LIN {X 0,Y 632.529,Z 1162.181,A -85,B 0,C 180,E1 6544.101,E2 6544.101} C_VEL
LIN {X 0,Y 629.019,Z 1204.643,A -85,B 0,C 180,E1 6550.428,E2 6550.428} C_VEL
LIN {X 0,Y 627.402,Z 1233.315,A -85,B 0,C 180,E1 6556.71,E2 6556.71} C_VEL
LIN {X 0,Y 626.919,Z 1250.593,A -85,B 0,C 180,E1 6563.045,E2 6563.045} C_VEL
LIN {X 0,Y 626.986,Z 1256.412,A -85,B 0,C 180,E1 6567.918,E2 6567.918} C_VEL
LIN {X 0,Y 627.218,Z 1255.317,A -85,B 0,C 180,E1 6573.469,E2 6573.469} C_VEL
LIN {X 0,Y 627.216,Z 1244.04,A -85,B 0,C 180,E1 6579.754,E2 6579.754} C_VEL
LIN {X 0,Y 628.041,Z 1219.84,A -85,B 0,C 180,E1 6586.5,E2 6586.5} C_VEL
LIN {X 0,Y 630.682,Z 1183.615,A -85,B 0,C 180,E1 6592.9,E2 6592.9} C_VEL
LIN {X 0,Y 635.527,Z 1132.969,A -85,B 0,C 180,E1 6599.124,E2 6599.124} C_VEL
LIN {X 0,Y 642.274,Z 1070.411,A -85,B 0,C 180,E1 6604.511,E2 6604.511} C_VEL
LIN {X 0,Y 649.326,Z 1000.53,A -85,B 0,C 180,E1 6608.612,E2 6608.612} C_VEL
LIN {X 0,Y 654.879,Z 926.452,A -85,B 0,C 180,E1 6611.351,E2 6611.351} C_VEL
LIN {X 0,Y 655.116,Z 892.167,A -85,B 0,C 180,E1 6612.26,E2 6612.26} C_VEL
LIN {X 0,Y 626.271,Z 839.06,A -85,B 0,C 180,E1 6615.936,E2 6615.936} C_VEL
LIN {X 0,Y 626.249,Z 839.06,A -85,B 0,C 180,E1 6624.3,E2 6624.3} C_VEL
LIN {X 0,Y 626.373,Z 839.06,A -85,B 0,C 180,E1 6632.206,E2 6632.206} C_VEL
LIN {X 0,Y 626.221,Z 839.06,A -85,B 0,C 180,E1 6640.951,E2 6640.951} C_VEL
LIN {X 0,Y 626.965,Z 839.06,A -85,B 0,C 180,E1 6649.584,E2 6649.584} C_VEL
LIN {X 0,Y 627.516,Z 839.06,A -85,B 0,C 180,E1 6659.347,E2 6659.347} C_VEL
LIN {X 0,Y 626.832,Z 839.06,A -85,B 0,C 180,E1 6667.69,E2 6667.69} C_VEL
LIN {X 0,Y 626.275,Z 839.06,A -85,B 0,C 180,E1 6676.766,E2 6676.766} C_VEL
LIN {X 0,Y 626.335,Z 839.06,A -85,B 0,C 180,E1 6685.126,E2 6685.126} C_VEL
LIN {X 0,Y 626.126,Z 839.06,A -85,B 0,C 180,E1 6693.229,E2 6693.229} C_VEL
LIN {X 0,Y 626.05,Z 839.06,A -85,B 0,C 180,E1 6701.847,E2 6701.847} C_VEL
LIN {X 0,Y 626.572,Z 841.021,A -85,B 0,C 180,E1 6703.843,E2 6703.843} C_VEL
LIN {X 0,Y 640.02,Z 863.387,A -85,B 0,C 180,E1 6705.418,E2 6705.418} C_VEL
LIN {X 0,Y 644.521,Z 885.503,A -85,B 0,C 180,E1 6706.146,E2 6706.146} C_VEL
LIN {X 0,Y 651.275,Z 900.392,A -85,B 0,C 180,E1 6706.954,E2 6706.954} C_VEL
LIN {X 0,Y 647.369,Z 977.205,A -85,B 0,C 180,E1 6708.756,E2 6708.756} C_VEL
LIN {X 0,Y 641.012,Z 1049.358,A -85,B 0,C 180,E1 6711.835,E2 6711.835} C_VEL
LIN {X 0,Y 633.382,Z 1117.843,A -85,B 0,C 180,E1 6716.34,E2 6716.34} C_VEL
LIN {X 0,Y 626.55,Z 1177.833,A -85,B 0,C 180,E1 6722.084,E2 6722.084} C_VEL
LIN {X 0,Y 621.952,Z 1224.147,A -85,B 0,C 180,E1 6728.397,E2 6728.397} C_VEL
LIN {X 0,Y 619.792,Z 1256.235,A -85,B 0,C 180,E1 6734.734,E2 6734.734} C_VEL
LIN {X 0,Y 619.023,Z 1276.005,A -85,B 0,C 180,E1 6740.828,E2 6740.828} C_VEL
LIN {X 0,Y 618.825,Z 1285.35,A -85,B 0,C 180,E1 6746.484,E2 6746.484} C_VEL
LIN {X 0,Y 618.751,Z 1286.379,A -85,B 0,C 180,E1 6752.11,E2 6752.11} C_VEL
LIN {X 0,Y 618.913,Z 1279.146,A -85,B 0,C 180,E1 6757.754,E2 6757.754} C_VEL
LIN {X 0,Y 619.502,Z 1261.052,A -85,B 0,C 180,E1 6764.027,E2 6764.027} C_VEL
LIN {X 0,Y 621.388,Z 1231.04,A -85,B 0,C 180,E1 6770.441,E2 6770.441} C_VEL
LIN {X 0,Y 625.557,Z 1187.146,A -85,B 0,C 180,E1 6776.825,E2 6776.825} C_VEL
LIN {X 0,Y 632.04,Z 1129.362,A -85,B 0,C 180,E1 6782.714,E2 6782.714} C_VEL
LIN {X 0,Y 639.563,Z 1062.77,A -85,B 0,C 180,E1 6787.421,E2 6787.421} C_VEL
LIN {X 0,Y 646.292,Z 992.668,A -85,B 0,C 180,E1 6790.706,E2 6790.706} C_VEL
LIN {X 0,Y 650.782,Z 919.257,A -85,B 0,C 180,E1 6792.72,E2 6792.72} C_VEL
LIN {X 0,Y 650.036,Z 895.654,A -85,B 0,C 180,E1 6793.232,E2 6793.232} C_VEL
LIN {X 0,Y 618.189,Z 839.06,A -85,B 0,C 180,E1 6797.021,E2 6797.021} C_VEL
LIN {X 0,Y 618.365,Z 839.06,A -85,B 0,C 180,E1 6805.331,E2 6805.331} C_VEL
LIN {X 0,Y 618.596,Z 839.06,A -85,B 0,C 180,E1 6813.607,E2 6813.607} C_VEL
LIN {X 0,Y 618.576,Z 839.06,A -85,B 0,C 180,E1 6823.575,E2 6823.575} C_VEL
LIN {X 0,Y 618.896,Z 839.06,A -85,B 0,C 180,E1 6832.211,E2 6832.211} C_VEL
LIN {X 0,Y 618.875,Z 839.06,A -85,B 0,C 180,E1 6840.662,E2 6840.662} C_VEL
LIN {X 0,Y 618.452,Z 839.06,A -85,B 0,C 180,E1 6849.135,E2 6849.135} C_VEL
LIN {X 0,Y 618.386,Z 839.06,A -85,B 0,C 180,E1 6856.346,E2 6856.346} C_VEL
LIN {X 0,Y 618.266,Z 839.06,A -85,B 0,C 180,E1 6865.387,E2 6865.387} C_VEL
LIN {X 0,Y 618.098,Z 839.06,A -85,B 0,C 180,E1 6873.476,E2 6873.476} C_VEL
LIN {X 0,Y 618.165,Z 839.06,A -85,B 0,C 180,E1 6882.395,E2 6882.395} C_VEL
LIN {X 0,Y 618.334,Z 840.427,A -85,B 0,C 180,E1 6883.456,E2 6883.456} C_VEL
LIN {X 0,Y 650.507,Z 899.763,A -85,B 0,C 180,E1 6887.454,E2 6887.454} C_VEL
LIN {X 0,Y 645.669,Z 969.285,A -85,B 0,C 180,E1 6889.502,E2 6889.502} C_VEL
LIN {X 0,Y 638.674,Z 1040.727,A -85,B 0,C 180,E1 6893.01,E2 6893.01} C_VEL
LIN {X 0,Y 631.057,Z 1107.355,A -85,B 0,C 180,E1 6897.944,E2 6897.944} C_VEL
LIN {X 0,Y 624.785,Z 1164.218,A -85,B 0,C 180,E1 6904.026,E2 6904.026} C_VEL
LIN {X 0,Y 621.153,Z 1205.493,A -85,B 0,C 180,E1 6910.33,E2 6910.33} C_VEL
LIN {X 0,Y 619.342,Z 1234.621,A -85,B 0,C 180,E1 6916.895,E2 6916.895} C_VEL
LIN {X 0,Y 618.993,Z 1250.188,A -85,B 0,C 180,E1 6922.736,E2 6922.736} C_VEL
LIN {X 0,Y 618.99,Z 1256.411,A -85,B 0,C 180,E1 6927.891,E2 6927.891} C_VEL
LIN {X 0,Y 619.195,Z 1255.317,A -85,B 0,C 180,E1 6933.514,E2 6933.514} C_VEL
LIN {X 0,Y 619.187,Z 1244.041,A -85,B 0,C 180,E1 6939.882,E2 6939.882} C_VEL
LIN {X 0,Y 620.112,Z 1221.406,A -85,B 0,C 180,E1 6946.351,E2 6946.351} C_VEL
LIN {X 0,Y 622.85,Z 1185.248,A -85,B 0,C 180,E1 6952.953,E2 6952.953} C_VEL
LIN {X 0,Y 628.001,Z 1134.743,A -85,B 0,C 180,E1 6959.309,E2 6959.309} C_VEL
LIN {X 0,Y 635.169,Z 1072.5,A -85,B 0,C 180,E1 6964.782,E2 6964.782} C_VEL
LIN {X 0,Y 642.527,Z 1004.298,A -85,B 0,C 180,E1 6968.883,E2 6968.883} C_VEL
LIN {X 0,Y 648.507,Z 930.181,A -85,B 0,C 180,E1 6971.721,E2 6971.721} C_VEL
LIN {X 0,Y 649.203,Z 895.835,A -85,B 0,C 180,E1 6972.652,E2 6972.652} C_VEL
LIN {X 0,Y 618.208,Z 839.06,A -85,B 0,C 180,E1 6976.602,E2 6976.602} C_VEL
LIN {X 0,Y 618.164,Z 839.06,A -85,B 0,C 180,E1 6985.356,E2 6985.356} C_VEL
LIN {X 0,Y 618.224,Z 839.06,A -85,B 0,C 180,E1 6993.675,E2 6993.675} C_VEL
LIN {X 0,Y 618.253,Z 839.06,A -85,B 0,C 180,E1 7002.179,E2 7002.179} C_VEL
LIN {X 0,Y 619.084,Z 839.06,A -85,B 0,C 180,E1 7010.875,E2 7010.875} C_VEL
LIN {X 0,Y 619.506,Z 839.06,A -85,B 0,C 180,E1 7019.339,E2 7019.339} C_VEL
LIN {X 0,Y 618.8,Z 839.06,A -85,B 0,C 180,E1 7027.791,E2 7027.791} C_VEL
LIN {X 0,Y 618.364,Z 839.06,A -85,B 0,C 180,E1 7036.431,E2 7036.431} C_VEL
LIN {X 0,Y 618.275,Z 839.06,A -85,B 0,C 180,E1 7045.476,E2 7045.476} C_VEL
LIN {X 0,Y 618.098,Z 839.06,A -85,B 0,C 180,E1 7053.573,E2 7053.573} C_VEL
LIN {X 0,Y 618.125,Z 839.06,A -85,B 0,C 180,E1 7062.508,E2 7062.508} C_VEL
LIN {X 0,Y 618.588,Z 841.588,A -85,B 0,C 180,E1 7063.083,E2 7063.083} C_VEL
LIN {X 0,Y 644.521,Z 885.503,A -85,B 0,C 180,E1 7066.146,E2 7066.146} C_VEL
LIN {X 0,Y 646.583,Z 902.081,A -85,B 0,C 180,E1 7066.594,E2 7066.594} C_VEL
LIN {X 0,Y 644.57,Z 920.711,A -85,B 0,C 180,E1 7066.802,E2 7066.802} C_VEL
LIN {X 0,Y 639.122,Z 999.805,A -85,B 0,C 180,E1 7069.069,E2 7069.069} C_VEL
LIN {X 0,Y 631.66,Z 1073.992,A -85,B 0,C 180,E1 7072.805,E2 7072.805} C_VEL
LIN {X 0,Y 623.945,Z 1139.278,A -85,B 0,C 180,E1 7077.768,E2 7077.768} C_VEL
LIN {X 0,Y 617.63,Z 1194.659,A -85,B 0,C 180,E1 7083.808,E2 7083.808} C_VEL
LIN {X 0,Y 613.673,Z 1237.403,A -85,B 0,C 180,E1 7090.491,E2 7090.491} C_VEL
LIN {X 0,Y 611.854,Z 1267.958,A -85,B 0,C 180,E1 7097.825,E2 7097.825} C_VEL
LIN {X 0,Y 611.014,Z 1283.797,A -85,B 0,C 180,E1 7105.012,E2 7105.012} C_VEL
LIN {X 0,Y 611.015,Z 1286.837,A -85,B 0,C 180,E1 7110.712,E2 7110.712} C_VEL
LIN {X 0,Y 610.942,Z 1280.509,A -85,B 0,C 180,E1 7117.138,E2 7117.138} C_VEL
LIN {X 0,Y 611.463,Z 1263.143,A -85,B 0,C 180,E1 7123.643,E2 7123.643} C_VEL
LIN {X 0,Y 613.267,Z 1234.809,A -85,B 0,C 180,E1 7130.019,E2 7130.019} C_VEL
LIN {X 0,Y 617.386,Z 1193.464,A -85,B 0,C 180,E1 7136.364,E2 7136.364} C_VEL
LIN {X 0,Y 624.114,Z 1136.467,A -85,B 0,C 180,E1 7142.497,E2 7142.497} C_VEL
LIN {X 0,Y 632.198,Z 1069.94,A -85,B 0,C 180,E1 7147.443,E2 7147.443} C_VEL
LIN {X 0,Y 639.445,Z 1000.576,A -85,B 0,C 180,E1 7150.87,E2 7150.87} C_VEL
LIN {X 0,Y 644.506,Z 926.944,A -85,B 0,C 180,E1 7153.057,E2 7153.057} C_VEL
LIN {X 0,Y 644.183,Z 899.082,A -85,B 0,C 180,E1 7153.661,E2 7153.661} C_VEL
LIN {X 0,Y 610.104,Z 839.06,A -85,B 0,C 180,E1 7157.851,E2 7157.851} C_VEL
LIN {X 0,Y 610.384,Z 839.06,A -85,B 0,C 180,E1 7166.429,E2 7166.429} C_VEL
LIN {X 0,Y 610.523,Z 839.06,A -85,B 0,C 180,E1 7175.177,E2 7175.177} C_VEL
LIN {X 0,Y 610.474,Z 839.06,A -85,B 0,C 180,E1 7184.831,E2 7184.831} C_VEL
LIN {X 0,Y 610.556,Z 839.06,A -85,B 0,C 180,E1 7193.539,E2 7193.539} C_VEL
LIN {X 0,Y 610.866,Z 839.06,A -85,B 0,C 180,E1 7200.671,E2 7200.671} C_VEL
LIN {X 0,Y 610.864,Z 839.06,A -85,B 0,C 180,E1 7207.81,E2 7207.81} C_VEL
LIN {X 0,Y 610.285,Z 839.06,A -85,B 0,C 180,E1 7216.721,E2 7216.721} C_VEL
LIN {X 0,Y 610.235,Z 839.06,A -85,B 0,C 180,E1 7225.746,E2 7225.746} C_VEL
LIN {X 0,Y 610.108,Z 839.06,A -85,B 0,C 180,E1 7233.973,E2 7233.973} C_VEL
LIN {X 0,Y 610.414,Z 840.999,A -85,B 0,C 180,E1 7242.67,E2 7242.67} C_VEL
LIN {X 0,Y 644.471,Z 901.549,A -85,B 0,C 180,E1 7247.003,E2 7247.003} C_VEL
LIN {X 0,Y 639.37,Z 970.596,A -85,B 0,C 180,E1 7249.08,E2 7249.08} C_VEL
LIN {X 0,Y 631.998,Z 1041.381,A -85,B 0,C 180,E1 7252.599,E2 7252.599} C_VEL
LIN {X 0,Y 623.815,Z 1108.393,A -85,B 0,C 180,E1 7257.629,E2 7257.629} C_VEL
LIN {X 0,Y 617.269,Z 1164.261,A -85,B 0,C 180,E1 7263.693,E2 7263.693} C_VEL
LIN {X 0,Y 613.256,Z 1206.563,A -85,B 0,C 180,E1 7270.271,E2 7270.271} C_VEL
LIN {X 0,Y 611.419,Z 1234.62,A -85,B 0,C 180,E1 7276.722,E2 7276.722} C_VEL
LIN {X 0,Y 611.016,Z 1250.187,A -85,B 0,C 180,E1 7282.641,E2 7282.641} C_VEL
LIN {X 0,Y 610.994,Z 1256.411,A -85,B 0,C 180,E1 7287.864,E2 7287.864} C_VEL
LIN {X 0,Y 611.174,Z 1255.317,A -85,B 0,C 180,E1 7293.56,E2 7293.56} C_VEL
LIN {X 0,Y 611.169,Z 1244.042,A -85,B 0,C 180,E1 7300.013,E2 7300.013} C_VEL
LIN {X 0,Y 612.17,Z 1221.41,A -85,B 0,C 180,E1 7306.57,E2 7306.57} C_VEL
LIN {X 0,Y 615.056,Z 1186.459,A -85,B 0,C 180,E1 7313.068,E2 7313.068} C_VEL
LIN {X 0,Y 620.57,Z 1135.75,A -85,B 0,C 180,E1 7319.58,E2 7319.58} C_VEL
LIN {X 0,Y 628.092,Z 1074.411,A -85,B 0,C 180,E1 7325.072,E2 7325.072} C_VEL
LIN {X 0,Y 635.917,Z 1006.392,A -85,B 0,C 180,E1 7329.244,E2 7329.244} C_VEL
LIN {X 0,Y 642.356,Z 932.017,A -85,B 0,C 180,E1 7332.149,E2 7332.149} C_VEL
LIN {X 0,Y 643.12,Z 899.03,A -85,B 0,C 180,E1 7333.078,E2 7333.078} C_VEL
LIN {X 0,Y 610.158,Z 839.06,A -85,B 0,C 180,E1 7337.417,E2 7337.417} C_VEL
LIN {X 0,Y 610.114,Z 839.06,A -85,B 0,C 180,E1 7346.466,E2 7346.466} C_VEL
LIN {X 0,Y 610.263,Z 839.06,A -85,B 0,C 180,E1 7355.228,E2 7355.228} C_VEL
LIN {X 0,Y 610.445,Z 839.06,A -85,B 0,C 180,E1 7363.435,E2 7363.435} C_VEL
LIN {X 0,Y 610.9,Z 839.06,A -85,B 0,C 180,E1 7372.19,E2 7372.19} C_VEL
LIN {X 0,Y 610.764,Z 839.06,A -85,B 0,C 180,E1 7380.753,E2 7380.753} C_VEL
LIN {X 0,Y 610.749,Z 839.06,A -85,B 0,C 180,E1 7387.894,E2 7387.894} C_VEL
LIN {X 0,Y 610.296,Z 839.06,A -85,B 0,C 180,E1 7396.728,E2 7396.728} C_VEL
LIN {X 0,Y 610.285,Z 839.06,A -85,B 0,C 180,E1 7404.776,E2 7404.776} C_VEL
LIN {X 0,Y 610.117,Z 839.06,A -85,B 0,C 180,E1 7413.535,E2 7413.535} C_VEL
LIN {X 0,Y 610.295,Z 840.83,A -85,B 0,C 180,E1 7422.238,E2 7422.238} C_VEL
LIN {X 0,Y 645.268,Z 901.082,A -85,B 0,C 180,E1 7426.466,E2 7426.466} C_VEL
LIN {X 0,Y 644.57,Z 920.711,A -85,B 0,C 180,E1 7426.802,E2 7426.802} C_VEL
LIN {X 0,Y 637.098,Z 955.226,A -85,B 0,C 180,E1 7427.137,E2 7427.137} C_VEL
LIN {X 0,Y 630.637,Z 1026.622,A -85,B 0,C 180,E1 7429.756,E2 7429.756} C_VEL
LIN {X 0,Y 622.159,Z 1097.78,A -85,B 0,C 180,E1 7433.945,E2 7433.945} C_VEL
LIN {X 0,Y 614.134,Z 1160.209,A -85,B 0,C 180,E1 7439.391,E2 7439.391} C_VEL
LIN {X 0,Y 608.038,Z 1211.489,A -85,B 0,C 180,E1 7445.807,E2 7445.807} C_VEL
LIN {X 0,Y 604.534,Z 1249.804,A -85,B 0,C 180,E1 7452.784,E2 7452.784} C_VEL
LIN {X 0,Y 603.318,Z 1272.228,A -85,B 0,C 180,E1 7459.122,E2 7459.122} C_VEL
LIN {X 0,Y 603.036,Z 1283.794,A -85,B 0,C 180,E1 7464.945,E2 7464.945} C_VEL
LIN {X 0,Y 603.01,Z 1286.837,A -85,B 0,C 180,E1 7470.722,E2 7470.722} C_VEL
LIN {X 0,Y 602.961,Z 1280.508,A -85,B 0,C 180,E1 7477.233,E2 7477.233} C_VEL
LIN {X 0,Y 603.513,Z 1263.143,A -85,B 0,C 180,E1 7483.826,E2 7483.826} C_VEL
LIN {X 0,Y 605.407,Z 1235.634,A -85,B 0,C 180,E1 7490.131,E2 7490.131} C_VEL
LIN {X 0,Y 609.837,Z 1193.617,A -85,B 0,C 180,E1 7496.695,E2 7496.695} C_VEL
LIN {X 0,Y 616.905,Z 1137.661,A -85,B 0,C 180,E1 7502.806,E2 7502.806} C_VEL
LIN {X 0,Y 625.495,Z 1071.067,A -85,B 0,C 180,E1 7507.834,E2 7507.834} C_VEL
LIN {X 0,Y 633.192,Z 1001.774,A -85,B 0,C 180,E1 7511.306,E2 7511.306} C_VEL
LIN {X 0,Y 638.628,Z 927.423,A -85,B 0,C 180,E1 7513.539,E2 7513.539} C_VEL
LIN {X 0,Y 638.377,Z 902.376,A -85,B 0,C 180,E1 7514.1,E2 7514.1} C_VEL
LIN {X 0,Y 602.069,Z 839.06,A -85,B 0,C 180,E1 7518.711,E2 7518.711} C_VEL
LIN {X 0,Y 602.468,Z 839.06,A -85,B 0,C 180,E1 7527.581,E2 7527.581} C_VEL
LIN {X 0,Y 602.512,Z 839.06,A -85,B 0,C 180,E1 7535.404,E2 7535.404} C_VEL
LIN {X 0,Y 602.456,Z 839.06,A -85,B 0,C 180,E1 7544.624,E2 7544.624} C_VEL
LIN {X 0,Y 602.594,Z 839.06,A -85,B 0,C 180,E1 7553.453,E2 7553.453} C_VEL
LIN {X 0,Y 602.858,Z 839.06,A -85,B 0,C 180,E1 7560.68,E2 7560.68} C_VEL
LIN {X 0,Y 602.831,Z 839.06,A -85,B 0,C 180,E1 7567.915,E2 7567.915} C_VEL
LIN {X 0,Y 602.28,Z 839.06,A -85,B 0,C 180,E1 7576.796,E2 7576.796} C_VEL
LIN {X 0,Y 602.317,Z 839.06,A -85,B 0,C 180,E1 7584.513,E2 7584.513} C_VEL
LIN {X 0,Y 602.127,Z 839.06,A -85,B 0,C 180,E1 7592.753,E2 7592.753} C_VEL
LIN {X 0,Y 602.079,Z 839.139,A -85,B 0,C 180,E1 7601.764,E2 7601.764} C_VEL
LIN {X 0,Y 638.349,Z 904.917,A -85,B 0,C 180,E1 7606.582,E2 7606.582} C_VEL
LIN {X 0,Y 632.904,Z 973.934,A -85,B 0,C 180,E1 7608.728,E2 7608.728} C_VEL
LIN {X 0,Y 625.101,Z 1044.237,A -85,B 0,C 180,E1 7612.319,E2 7612.319} C_VEL
LIN {X 0,Y 616.454,Z 1110.841,A -85,B 0,C 180,E1 7617.438,E2 7617.438} C_VEL
LIN {X 0,Y 609.485,Z 1166.513,A -85,B 0,C 180,E1 7623.638,E2 7623.638} C_VEL
LIN {X 0,Y 605.361,Z 1207.623,A -85,B 0,C 180,E1 7630.211,E2 7630.211} C_VEL
LIN {X 0,Y 603.395,Z 1235.781,A -85,B 0,C 180,E1 7636.912,E2 7636.912} C_VEL
LIN {X 0,Y 602.915,Z 1251.796,A -85,B 0,C 180,E1 7643.494,E2 7643.494} C_VEL
LIN {X 0,Y 602.68,Z 1256.848,A -85,B 0,C 180,E1 7649.278,E2 7649.278} C_VEL
LIN {X 0,Y 602.912,Z 1252.806,A -85,B 0,C 180,E1 7655.78,E2 7655.78} C_VEL
LIN {X 0,Y 603.585,Z 1236.661,A -85,B 0,C 180,E1 7662.713,E2 7662.713} C_VEL
LIN {X 0,Y 605.898,Z 1205.828,A -85,B 0,C 180,E1 7670.032,E2 7670.032} C_VEL
LIN {X 0,Y 610.609,Z 1160.875,A -85,B 0,C 180,E1 7676.987,E2 7676.987} C_VEL
LIN {X 0,Y 617.438,Z 1104.611,A -85,B 0,C 180,E1 7683.033,E2 7683.033} C_VEL
LIN {X 0,Y 625.742,Z 1038.363,A -85,B 0,C 180,E1 7687.965,E2 7687.965} C_VEL
LIN {X 0,Y 633.664,Z 964.987,A -85,B 0,C 180,E1 7691.542,E2 7691.542} C_VEL
LIN {X 0,Y 637.241,Z 902.506,A -85,B 0,C 180,E1 7693.491,E2 7693.491} C_VEL
LIN {X 0,Y 603.882,Z 844.033,A -85,B 0,C 180,E1 7697.868,E2 7697.868} C_VEL
LIN {X 0,Y 602.111,Z 839.06,A -85,B 0,C 180,E1 7698.163,E2 7698.163} C_VEL
LIN {X 0,Y 602.125,Z 839.06,A -85,B 0,C 180,E1 7707.247,E2 7707.247} C_VEL
LIN {X 0,Y 602.303,Z 839.06,A -85,B 0,C 180,E1 7715.486,E2 7715.486} C_VEL
LIN {X 0,Y 602.666,Z 839.06,A -85,B 0,C 180,E1 7724.716,E2 7724.716} C_VEL
LIN {X 0,Y 602.908,Z 839.06,A -85,B 0,C 180,E1 7732.086,E2 7732.086} C_VEL
LIN {X 0,Y 602.758,Z 839.06,A -85,B 0,C 180,E1 7740.763,E2 7740.763} C_VEL
LIN {X 0,Y 602.699,Z 839.06,A -85,B 0,C 180,E1 7748,E2 7748} C_VEL
LIN {X 0,Y 602.278,Z 839.06,A -85,B 0,C 180,E1 7756.883,E2 7756.883} C_VEL
LIN {X 0,Y 602.3,Z 839.06,A -85,B 0,C 180,E1 7764.605,E2 7764.605} C_VEL
LIN {X 0,Y 602.121,Z 839.06,A -85,B 0,C 180,E1 7772.852,E2 7772.852} C_VEL
LIN {X 0,Y 602.239,Z 840.755,A -85,B 0,C 180,E1 7781.393,E2 7781.393} C_VEL
LIN {X 0,Y 639.23,Z 904.05,A -85,B 0,C 180,E1 7786.005,E2 7786.005} C_VEL
LIN {X 0,Y 637.098,Z 955.226,A -85,B 0,C 180,E1 7787.137,E2 7787.137} C_VEL
LIN {X 0,Y 628.191,Z 989.03,A -85,B 0,C 180,E1 7787.698,E2 7787.698} C_VEL
LIN {X 0,Y 620.228,Z 1061.943,A -85,B 0,C 180,E1 7791.144,E2 7791.144} C_VEL
LIN {X 0,Y 611.113,Z 1129.374,A -85,B 0,C 180,E1 7796.018,E2 7796.018} C_VEL
LIN {X 0,Y 603.289,Z 1187.108,A -85,B 0,C 180,E1 7802.094,E2 7802.094} C_VEL
LIN {X 0,Y 598.231,Z 1232.469,A -85,B 0,C 180,E1 7808.996,E2 7808.996} C_VEL
LIN {X 0,Y 596.057,Z 1264.475,A -85,B 0,C 180,E1 7816.374,E2 7816.374} C_VEL
LIN {X 0,Y 595.5,Z 1281.719,A -85,B 0,C 180,E1 7823.413,E2 7823.413} C_VEL
LIN {X 0,Y 595.032,Z 1286.837,A -85,B 0,C 180,E1 7830.731,E2 7830.731} C_VEL
LIN {X 0,Y 594.977,Z 1280.505,A -85,B 0,C 180,E1 7837.33,E2 7837.33} C_VEL
LIN {X 0,Y 595.579,Z 1263.142,A -85,B 0,C 180,E1 7844.014,E2 7844.014} C_VEL
LIN {X 0,Y 597.651,Z 1235.436,A -85,B 0,C 180,E1 7850.443,E2 7850.443} C_VEL
LIN {X 0,Y 602.302,Z 1193.887,A -85,B 0,C 180,E1 7857.018,E2 7857.018} C_VEL
LIN {X 0,Y 609.977,Z 1137.087,A -85,B 0,C 180,E1 7863.284,E2 7863.284} C_VEL
LIN {X 0,Y 618.981,Z 1071.107,A -85,B 0,C 180,E1 7868.301,E2 7868.301} C_VEL
LIN {X 0,Y 627.135,Z 1001.143,A -85,B 0,C 180,E1 7871.824,E2 7871.824} C_VEL
LIN {X 0,Y 632.778,Z 928.03,A -85,B 0,C 180,E1 7874.028,E2 7874.028} C_VEL
LIN {X 0,Y 632.297,Z 905.261,A -85,B 0,C 180,E1 7874.578,E2 7874.578} C_VEL
LIN {X 0,Y 596.01,Z 844.293,A -85,B 0,C 180,E1 7879.222,E2 7879.222} C_VEL
LIN {X 0,Y 594.085,Z 839.06,A -85,B 0,C 180,E1 7879.61,E2 7879.61} C_VEL
LIN {X 0,Y 594.467,Z 839.06,A -85,B 0,C 180,E1 7888.816,E2 7888.816} C_VEL
LIN {X 0,Y 594.331,Z 839.06,A -85,B 0,C 180,E1 7896.646,E2 7896.646} C_VEL
LIN {X 0,Y 594.359,Z 839.06,A -85,B 0,C 180,E1 7905.922,E2 7905.922} C_VEL
LIN {X 0,Y 594.602,Z 839.06,A -85,B 0,C 180,E1 7913.364,E2 7913.364} C_VEL
LIN {X 0,Y 594.849,Z 839.06,A -85,B 0,C 180,E1 7920.689,E2 7920.689} C_VEL
LIN {X 0,Y 594.782,Z 839.06,A -85,B 0,C 180,E1 7928.023,E2 7928.023} C_VEL
LIN {X 0,Y 594.225,Z 839.06,A -85,B 0,C 180,E1 7937.031,E2 7937.031} C_VEL
LIN {X 0,Y 594.243,Z 839.06,A -85,B 0,C 180,E1 7944.916,E2 7944.916} C_VEL
LIN {X 0,Y 594.024,Z 839.06,A -85,B 0,C 180,E1 7953.84,E2 7953.84} C_VEL
LIN {X 0,Y 594.3,Z 840.985,A -85,B 0,C 180,E1 7960.944,E2 7960.944} C_VEL
LIN {X 0,Y 628.756,Z 900.689,A -85,B 0,C 180,E1 7965.629,E2 7965.629} C_VEL
LIN {X 0,Y 632.023,Z 912.179,A -85,B 0,C 180,E1 7966.257,E2 7966.257} C_VEL
LIN {X 0,Y 626.061,Z 981.748,A -85,B 0,C 180,E1 7968.558,E2 7968.558} C_VEL
LIN {X 0,Y 617.713,Z 1050.945,A -85,B 0,C 180,E1 7972.276,E2 7972.276} C_VEL
LIN {X 0,Y 608.668,Z 1116.732,A -85,B 0,C 180,E1 7977.571,E2 7977.571} C_VEL
LIN {X 0,Y 601.336,Z 1171.593,A -85,B 0,C 180,E1 7983.982,E2 7983.982} C_VEL
LIN {X 0,Y 597.151,Z 1211.506,A -85,B 0,C 180,E1 7990.701,E2 7990.701} C_VEL
LIN {X 0,Y 595.367,Z 1236.942,A -85,B 0,C 180,E1 7997.108,E2 7997.108} C_VEL
LIN {X 0,Y 594.938,Z 1251.792,A -85,B 0,C 180,E1 8003.406,E2 8003.406} C_VEL
LIN {X 0,Y 594.681,Z 1256.848,A -85,B 0,C 180,E1 8009.268,E2 8009.268} C_VEL
LIN {X 0,Y 594.939,Z 1252.807,A -85,B 0,C 180,E1 8015.858,E2 8015.858} C_VEL
LIN {X 0,Y 595.685,Z 1236.664,A -85,B 0,C 180,E1 8022.885,E2 8022.885} C_VEL
LIN {X 0,Y 598.162,Z 1205.829,A -85,B 0,C 180,E1 8030.303,E2 8030.303} C_VEL
LIN {X 0,Y 603.221,Z 1160.195,A -85,B 0,C 180,E1 8037.44,E2 8037.44} C_VEL
LIN {X 0,Y 610.695,Z 1102.99,A -85,B 0,C 180,E1 8043.61,E2 8043.61} C_VEL
LIN {X 0,Y 619.491,Z 1036.605,A -85,B 0,C 180,E1 8048.546,E2 8048.546} C_VEL
LIN {X 0,Y 627.757,Z 963.177,A -85,B 0,C 180,E1 8052.108,E2 8052.108} C_VEL
LIN {X 0,Y 631.077,Z 905.613,A -85,B 0,C 180,E1 8053.936,E2 8053.936} C_VEL
LIN {X 0,Y 599.364,Z 849.392,A -85,B 0,C 180,E1 8058.257,E2 8058.257} C_VEL
LIN {X 0,Y 594.03,Z 839.06,A -85,B 0,C 180,E1 8059.198,E2 8059.198} C_VEL
LIN {X 0,Y 594.219,Z 839.06,A -85,B 0,C 180,E1 8068.488,E2 8068.488} C_VEL
LIN {X 0,Y 594.377,Z 839.06,A -85,B 0,C 180,E1 8076.739,E2 8076.739} C_VEL
LIN {X 0,Y 594.782,Z 839.06,A -85,B 0,C 180,E1 8086.019,E2 8086.019} C_VEL
LIN {X 0,Y 594.567,Z 839.06,A -85,B 0,C 180,E1 8093.449,E2 8093.449} C_VEL
LIN {X 0,Y 594.756,Z 839.06,A -85,B 0,C 180,E1 8100.773,E2 8100.773} C_VEL
LIN {X 0,Y 594.653,Z 839.06,A -85,B 0,C 180,E1 8108.109,E2 8108.109} C_VEL
LIN {X 0,Y 594.253,Z 839.06,A -85,B 0,C 180,E1 8117.118,E2 8117.118} C_VEL
LIN {X 0,Y 594.253,Z 839.06,A -85,B 0,C 180,E1 8124.961,E2 8124.961} C_VEL
LIN {X 0,Y 594.031,Z 839.06,A -85,B 0,C 180,E1 8133.843,E2 8133.843} C_VEL
LIN {X 0,Y 594.253,Z 840.855,A -85,B 0,C 180,E1 8140.521,E2 8140.521} C_VEL
LIN {X 0,Y 633.142,Z 906.971,A -85,B 0,C 180,E1 8145.528,E2 8145.528} C_VEL
LIN {X 0,Y 628.46,Z 986.241,A -85,B 0,C 180,E1 8147.604,E2 8147.604} C_VEL
LIN {X 0,Y 628.191,Z 989.03,A -85,B 0,C 180,E1 8147.698,E2 8147.698} C_VEL
LIN {X 0,Y 619.77,Z 1011.161,A -85,B 0,C 180,E1 8148.057,E2 8148.057} C_VEL
LIN {X 0,Y 610.69,Z 1083.868,A -85,B 0,C 180,E1 8152.038,E2 8152.038} C_VEL
LIN {X 0,Y 601.535,Z 1148.423,A -85,B 0,C 180,E1 8157.373,E2 8157.373} C_VEL
LIN {X 0,Y 594.154,Z 1202.648,A -85,B 0,C 180,E1 8163.849,E2 8163.849} C_VEL
LIN {X 0,Y 589.634,Z 1244.839,A -85,B 0,C 180,E1 8171.227,E2 8171.227} C_VEL
LIN {X 0,Y 587.441,Z 1272.229,A -85,B 0,C 180,E1 8178.825,E2 8178.825} C_VEL
LIN {X 0,Y 587.081,Z 1283.788,A -85,B 0,C 180,E1 8184.808,E2 8184.808} C_VEL
LIN {X 0,Y 587.027,Z 1286.837,A -85,B 0,C 180,E1 8190.741,E2 8190.741} C_VEL
LIN {X 0,Y 586.975,Z 1280.502,A -85,B 0,C 180,E1 8197.431,E2 8197.431} C_VEL
LIN {X 0,Y 587.657,Z 1263.141,A -85,B 0,C 180,E1 8204.207,E2 8204.207} C_VEL
LIN {X 0,Y 590.07,Z 1233.454,A -85,B 0,C 180,E1 8211.112,E2 8211.112} C_VEL
LIN {X 0,Y 595.727,Z 1188.276,A -85,B 0,C 180,E1 8218.129,E2 8218.129} C_VEL
LIN {X 0,Y 604.023,Z 1130.665,A -85,B 0,C 180,E1 8224.314,E2 8224.314} C_VEL
LIN {X 0,Y 613.535,Z 1063.651,A -85,B 0,C 180,E1 8229.246,E2 8229.246} C_VEL
LIN {X 0,Y 621.894,Z 993.828,A -85,B 0,C 180,E1 8232.612,E2 8232.612} C_VEL
LIN {X 0,Y 627.33,Z 922.424,A -85,B 0,C 180,E1 8234.643,E2 8234.643} C_VEL
LIN {X 0,Y 626.266,Z 908.039,A -85,B 0,C 180,E1 8235.067,E2 8235.067} C_VEL
LIN {X 0,Y 588.791,Z 845.036,A -85,B 0,C 180,E1 8240.024,E2 8240.024} C_VEL
LIN {X 0,Y 586.171,Z 839.06,A -85,B 0,C 180,E1 8240.589,E2 8240.589} C_VEL
LIN {X 0,Y 586.447,Z 839.06,A -85,B 0,C 180,E1 8250.136,E2 8250.136} C_VEL
LIN {X 0,Y 586.125,Z 839.06,A -85,B 0,C 180,E1 8257.909,E2 8257.909} C_VEL
LIN {X 0,Y 586.332,Z 839.06,A -85,B 0,C 180,E1 8266.155,E2 8266.155} C_VEL
LIN {X 0,Y 586.622,Z 839.06,A -85,B 0,C 180,E1 8273.274,E2 8273.274} C_VEL
LIN {X 0,Y 586.841,Z 839.06,A -85,B 0,C 180,E1 8280.698,E2 8280.698} C_VEL
LIN {X 0,Y 586.735,Z 839.06,A -85,B 0,C 180,E1 8288.133,E2 8288.133} C_VEL
LIN {X 0,Y 586.178,Z 839.06,A -85,B 0,C 180,E1 8297.272,E2 8297.272} C_VEL
LIN {X 0,Y 586.227,Z 839.06,A -85,B 0,C 180,E1 8305.232,E2 8305.232} C_VEL
LIN {X 0,Y 586.043,Z 839.06,A -85,B 0,C 180,E1 8313.77,E2 8313.77} C_VEL
LIN {X 0,Y 586.133,Z 840.441,A -85,B 0,C 180,E1 8319.999,E2 8319.999} C_VEL
LIN {X 0,Y 621.646,Z 901.479,A -85,B 0,C 180,E1 8324.997,E2 8324.997} C_VEL
LIN {X 0,Y 626.079,Z 914.944,A -85,B 0,C 180,E1 8325.812,E2 8325.812} C_VEL
LIN {X 0,Y 619.684,Z 984.03,A -85,B 0,C 180,E1 8328.162,E2 8328.162} C_VEL
LIN {X 0,Y 610.83,Z 1053.59,A -85,B 0,C 180,E1 8331.98,E2 8331.98} C_VEL
LIN {X 0,Y 601.338,Z 1118.473,A -85,B 0,C 180,E1 8337.321,E2 8337.321} C_VEL
LIN {X 0,Y 593.627,Z 1172.937,A -85,B 0,C 180,E1 8343.823,E2 8343.823} C_VEL
LIN {X 0,Y 589.327,Z 1211.681,A -85,B 0,C 180,E1 8350.473,E2 8350.473} C_VEL
LIN {X 0,Y 587.441,Z 1236.94,A -85,B 0,C 180,E1 8356.93,E2 8356.93} C_VEL
LIN {X 0,Y 586.961,Z 1251.788,A -85,B 0,C 180,E1 8363.316,E2 8363.316} C_VEL
LIN {X 0,Y 586.683,Z 1256.848,A -85,B 0,C 180,E1 8369.258,E2 8369.258} C_VEL
LIN {X 0,Y 586.881,Z 1253.736,A -85,B 0,C 180,E1 8375.194,E2 8375.194} C_VEL
LIN {X 0,Y 587.32,Z 1240.12,A -85,B 0,C 180,E1 8381.934,E2 8381.934} C_VEL
LIN {X 0,Y 589.119,Z 1214.638,A -85,B 0,C 180,E1 8388.79,E2 8388.79} C_VEL
LIN {X 0,Y 593.541,Z 1175.015,A -85,B 0,C 180,E1 8395.773,E2 8395.773} C_VEL
LIN {X 0,Y 600.98,Z 1120.999,A -85,B 0,C 180,E1 8402.329,E2 8402.329} C_VEL
LIN {X 0,Y 610.333,Z 1056.636,A -85,B 0,C 180,E1 8407.719,E2 8407.719} C_VEL
LIN {X 0,Y 619.42,Z 986.417,A -85,B 0,C 180,E1 8411.639,E2 8411.639} C_VEL
LIN {X 0,Y 626.039,Z 916.562,A -85,B 0,C 180,E1 8414.052,E2 8414.052} C_VEL
LIN {X 0,Y 622.509,Z 903.37,A -85,B 0,C 180,E1 8414.784,E2 8414.784} C_VEL
LIN {X 0,Y 589.079,Z 845.345,A -85,B 0,C 180,E1 8419.476,E2 8419.476} C_VEL
LIN {X 0,Y 586.009,Z 839.06,A -85,B 0,C 180,E1 8420.29,E2 8420.29} C_VEL
LIN {X 0,Y 586.25,Z 839.06,A -85,B 0,C 180,E1 8429.741,E2 8429.741} C_VEL
LIN {X 0,Y 586.344,Z 839.06,A -85,B 0,C 180,E1 8438.01,E2 8438.01} C_VEL
LIN {X 0,Y 586.75,Z 839.06,A -85,B 0,C 180,E1 8447.347,E2 8447.347} C_VEL
LIN {X 0,Y 586.384,Z 839.06,A -85,B 0,C 180,E1 8455.37,E2 8455.37} C_VEL
LIN {X 0,Y 586.75,Z 839.06,A -85,B 0,C 180,E1 8460.783,E2 8460.783} C_VEL
LIN {X 0,Y 586.608,Z 839.06,A -85,B 0,C 180,E1 8468.221,E2 8468.221} C_VEL
LIN {X 0,Y 586.199,Z 839.06,A -85,B 0,C 180,E1 8477.361,E2 8477.361} C_VEL
LIN {X 0,Y 586.203,Z 839.06,A -85,B 0,C 180,E1 8485.327,E2 8485.327} C_VEL
LIN {X 0,Y 586.029,Z 839.06,A -85,B 0,C 180,E1 8493.874,E2 8493.874} C_VEL
LIN {X 0,Y 586.321,Z 840.939,A -85,B 0,C 180,E1 8499.615,E2 8499.615} C_VEL
LIN {X 0,Y 624.852,Z 905.465,A -85,B 0,C 180,E1 8504.755,E2 8504.755} C_VEL
LIN {X 0,Y 627.452,Z 915.546,A -85,B 0,C 180,E1 8505.199,E2 8505.199} C_VEL
LIN {X 0,Y 621.618,Z 993.895,A -85,B 0,C 180,E1 8507.367,E2 8507.367} C_VEL
LIN {X 0,Y 619.77,Z 1011.161,A -85,B 0,C 180,E1 8508.057,E2 8508.057} C_VEL
LIN {X 0,Y 609.963,Z 1043.36,A -85,B 0,C 180,E1 8509.12,E2 8509.12} C_VEL
LIN {X 0,Y 600.01,Z 1111.635,A -85,B 0,C 180,E1 8513.619,E2 8513.619} C_VEL
LIN {X 0,Y 590.55,Z 1173,A -85,B 0,C 180,E1 8519.591,E2 8519.591} C_VEL
LIN {X 0,Y 583.889,Z 1221.503,A -85,B 0,C 180,E1 8526.429,E2 8526.429} C_VEL
LIN {X 0,Y 580.379,Z 1254.894,A -85,B 0,C 180,E1 8533.33,E2 8533.33} C_VEL
LIN {X 0,Y 579.111,Z 1276.005,A -85,B 0,C 180,E1 8540.19,E2 8540.19} C_VEL
LIN {X 0,Y 578.868,Z 1285.349,A -85,B 0,C 180,E1 8546.241,E2 8546.241} C_VEL
LIN {X 0,Y 578.82,Z 1286.379,A -85,B 0,C 180,E1 8552.255,E2 8552.255} C_VEL
LIN {X 0,Y 579.238,Z 1277.595,A -85,B 0,C 180,E1 8559.048,E2 8559.048} C_VEL
LIN {X 0,Y 580.977,Z 1254.689,A -85,B 0,C 180,E1 8566.705,E2 8566.705} C_VEL
LIN {X 0,Y 584.821,Z 1217.061,A -85,B 0,C 180,E1 8574.28,E2 8574.28} C_VEL
LIN {X 0,Y 591.822,Z 1165.647,A -85,B 0,C 180,E1 8581.232,E2 8581.232} C_VEL
LIN {X 0,Y 601.152,Z 1104.516,A -85,B 0,C 180,E1 8586.934,E2 8586.934} C_VEL
LIN {X 0,Y 610.899,Z 1034.056,A -85,B 0,C 180,E1 8591.38,E2 8591.38} C_VEL
LIN {X 0,Y 618.936,Z 957.216,A -85,B 0,C 180,E1 8594.351,E2 8594.351} C_VEL
LIN {X 0,Y 620.815,Z 912.065,A -85,B 0,C 180,E1 8595.491,E2 8595.491} C_VEL
LIN {X 0,Y 584.529,Z 850.775,A -85,B 0,C 180,E1 8600.413,E2 8600.413} C_VEL
LIN {X 0,Y 578.113,Z 839.06,A -85,B 0,C 180,E1 8601.558,E2 8601.558} C_VEL
LIN {X 0,Y 578.458,Z 839.06,A -85,B 0,C 180,E1 8610.924,E2 8610.924} C_VEL
LIN {X 0,Y 578.021,Z 839.06,A -85,B 0,C 180,E1 8619.2,E2 8619.2} C_VEL
LIN {X 0,Y 578.272,Z 839.06,A -85,B 0,C 180,E1 8627.07,E2 8627.07} C_VEL
LIN {X 0,Y 578.386,Z 839.06,A -85,B 0,C 180,E1 8634.689,E2 8634.689} C_VEL
LIN {X 0,Y 578.833,Z 839.06,A -85,B 0,C 180,E1 8640.708,E2 8640.708} C_VEL
LIN {X 0,Y 578.691,Z 839.06,A -85,B 0,C 180,E1 8648.247,E2 8648.247} C_VEL
LIN {X 0,Y 578.164,Z 839.06,A -85,B 0,C 180,E1 8657.519,E2 8657.519} C_VEL
LIN {X 0,Y 578.193,Z 839.06,A -85,B 0,C 180,E1 8665.608,E2 8665.608} C_VEL
LIN {X 0,Y 578.016,Z 839.06,A -85,B 0,C 180,E1 8674.304,E2 8674.304} C_VEL
LIN {X 0,Y 578.209,Z 840.785,A -85,B 0,C 180,E1 8679.053,E2 8679.053} C_VEL
LIN {X 0,Y 615.112,Z 903.174,A -85,B 0,C 180,E1 8684.422,E2 8684.422} C_VEL
LIN {X 0,Y 620.082,Z 918.824,A -85,B 0,C 180,E1 8685.385,E2 8685.385} C_VEL
LIN {X 0,Y 613.08,Z 988.633,A -85,B 0,C 180,E1 8687.861,E2 8687.861} C_VEL
LIN {X 0,Y 603.856,Z 1056.414,A -85,B 0,C 180,E1 8691.695,E2 8691.695} C_VEL
LIN {X 0,Y 594.008,Z 1120.207,A -85,B 0,C 180,E1 8697.064,E2 8697.064} C_VEL
LIN {X 0,Y 585.909,Z 1174.336,A -85,B 0,C 180,E1 8703.67,E2 8703.67} C_VEL
LIN {X 0,Y 581.318,Z 1213.498,A -85,B 0,C 180,E1 8710.602,E2 8710.602} C_VEL
LIN {X 0,Y 579.413,Z 1238.088,A -85,B 0,C 180,E1 8717.131,E2 8717.131} C_VEL
LIN {X 0,Y 578.948,Z 1252.778,A -85,B 0,C 180,E1 8723.868,E2 8723.868} C_VEL
LIN {X 0,Y 579.036,Z 1256.827,A -85,B 0,C 180,E1 8730.751,E2 8730.751} C_VEL
LIN {X 0,Y 579.473,Z 1249.059,A -85,B 0,C 180,E1 8738.284,E2 8738.284} C_VEL
LIN {X 0,Y 580.412,Z 1227.584,A -85,B 0,C 180,E1 8745.94,E2 8745.94} C_VEL
LIN {X 0,Y 583.884,Z 1191.855,A -85,B 0,C 180,E1 8753.466,E2 8753.466} C_VEL
LIN {X 0,Y 590.669,Z 1142.33,A -85,B 0,C 180,E1 8760.439,E2 8760.439} C_VEL
LIN {X 0,Y 600.125,Z 1081.182,A -85,B 0,C 180,E1 8766.368,E2 8766.368} C_VEL
LIN {X 0,Y 609.925,Z 1013.604,A -85,B 0,C 180,E1 8770.823,E2 8770.823} C_VEL
LIN {X 0,Y 618.161,Z 939.664,A -85,B 0,C 180,E1 8773.945,E2 8773.945} C_VEL
LIN {X 0,Y 619.092,Z 912.151,A -85,B 0,C 180,E1 8774.827,E2 8774.827} C_VEL
LIN {X 0,Y 589.037,Z 857.554,A -85,B 0,C 180,E1 8779.256,E2 8779.256} C_VEL
LIN {X 0,Y 578.017,Z 839.06,A -85,B 0,C 180,E1 8781.022,E2 8781.022} C_VEL
LIN {X 0,Y 578.161,Z 839.06,A -85,B 0,C 180,E1 8789.272,E2 8789.272} C_VEL
LIN {X 0,Y 578.279,Z 839.06,A -85,B 0,C 180,E1 8798.741,E2 8798.741} C_VEL
LIN {X 0,Y 578.738,Z 839.06,A -85,B 0,C 180,E1 8807.169,E2 8807.169} C_VEL
LIN {X 0,Y 578.391,Z 839.06,A -85,B 0,C 180,E1 8814.776,E2 8814.776} C_VEL
LIN {X 0,Y 578.743,Z 839.06,A -85,B 0,C 180,E1 8820.794,E2 8820.794} C_VEL
LIN {X 0,Y 578.567,Z 839.06,A -85,B 0,C 180,E1 8828.336,E2 8828.336} C_VEL
LIN {X 0,Y 578.153,Z 839.06,A -85,B 0,C 180,E1 8837.61,E2 8837.61} C_VEL
LIN {X 0,Y 578.187,Z 839.06,A -85,B 0,C 180,E1 8845.704,E2 8845.704} C_VEL
LIN {X 0,Y 578.006,Z 839.06,A -85,B 0,C 180,E1 8854.409,E2 8854.409} C_VEL
LIN {X 0,Y 578.251,Z 840.776,A -85,B 0,C 180,E1 8858.645,E2 8858.645} C_VEL
LIN {X 0,Y 618.048,Z 906.725,A -85,B 0,C 180,E1 8864.146,E2 8864.146} C_VEL
LIN {X 0,Y 621.59,Z 918.098,A -85,B 0,C 180,E1 8864.731,E2 8864.731} C_VEL
LIN {X 0,Y 615.228,Z 996.937,A -85,B 0,C 180,E1 8866.98,E2 8866.98} C_VEL
LIN {X 0,Y 609.963,Z 1043.36,A -85,B 0,C 180,E1 8869.12,E2 8869.12} C_VEL
LIN {X 0,Y 599.208,Z 1074.248,A -85,B 0,C 180,E1 8870.432,E2 8870.432} C_VEL
LIN {X 0,Y 588.862,Z 1139.399,A -85,B 0,C 180,E1 8875.603,E2 8875.603} C_VEL
LIN {X 0,Y 579.974,Z 1195.707,A -85,B 0,C 180,E1 8882.116,E2 8882.116} C_VEL
LIN {X 0,Y 574.377,Z 1239.427,A -85,B 0,C 180,E1 8889.517,E2 8889.517} C_VEL
LIN {X 0,Y 572.071,Z 1269.105,A -85,B 0,C 180,E1 8897.354,E2 8897.354} C_VEL
LIN {X 0,Y 571.15,Z 1283.782,A -85,B 0,C 180,E1 8904.663,E2 8904.663} C_VEL
LIN {X 0,Y 571.017,Z 1286.837,A -85,B 0,C 180,E1 8910.762,E2 8910.762} C_VEL
LIN {X 0,Y 571.016,Z 1280.497,A -85,B 0,C 180,E1 8917.639,E2 8917.639} C_VEL
LIN {X 0,Y 571.847,Z 1263.139,A -85,B 0,C 180,E1 8924.608,E2 8924.608} C_VEL
LIN {X 0,Y 574.835,Z 1232.465,A -85,B 0,C 180,E1 8931.903,E2 8931.903} C_VEL
LIN {X 0,Y 581.353,Z 1186.778,A -85,B 0,C 180,E1 8939.102,E2 8939.102} C_VEL
LIN {X 0,Y 590.693,Z 1128.305,A -85,B 0,C 180,E1 8945.433,E2 8945.433} C_VEL
LIN {X 0,Y 601.146,Z 1061.516,A -85,B 0,C 180,E1 8950.365,E2 8950.365} C_VEL
LIN {X 0,Y 610.36,Z 989.66,A -85,B 0,C 180,E1 8953.793,E2 8953.793} C_VEL
LIN {X 0,Y 615.038,Z 915.352,A -85,B 0,C 180,E1 8955.951,E2 8955.951} C_VEL
LIN {X 0,Y 577.827,Z 852.071,A -85,B 0,C 180,E1 8961.192,E2 8961.192} C_VEL
LIN {X 0,Y 570.114,Z 839.06,A -85,B 0,C 180,E1 8962.607,E2 8962.607} C_VEL
LIN {X 0,Y 570.381,Z 839.06,A -85,B 0,C 180,E1 8970.472,E2 8970.472} C_VEL
LIN {X 0,Y 570.048,Z 839.06,A -85,B 0,C 180,E1 8978.896,E2 8978.896} C_VEL
LIN {X 0,Y 570.261,Z 839.06,A -85,B 0,C 180,E1 8986.885,E2 8986.885} C_VEL
LIN {X 0,Y 570.391,Z 839.06,A -85,B 0,C 180,E1 8994.614,E2 8994.614} C_VEL
LIN {X 0,Y 570.825,Z 839.06,A -85,B 0,C 180,E1 9000.718,E2 9000.718} C_VEL
LIN {X 0,Y 570.669,Z 839.06,A -85,B 0,C 180,E1 9008.364,E2 9008.364} C_VEL
LIN {X 0,Y 570.125,Z 839.06,A -85,B 0,C 180,E1 9017.774,E2 9017.774} C_VEL
LIN {X 0,Y 570.135,Z 839.06,A -85,B 0,C 180,E1 9026.871,E2 9026.871} C_VEL
LIN {X 0,Y 569.959,Z 839.06,A -85,B 0,C 180,E1 9035.67,E2 9035.67} C_VEL
LIN {X 0,Y 570.229,Z 840.753,A -85,B 0,C 180,E1 9038.046,E2 9038.046} C_VEL
LIN {X 0,Y 608.1,Z 903.984,A -85,B 0,C 180,E1 9043.758,E2 9043.758} C_VEL
LIN {X 0,Y 614.132,Z 922.304,A -85,B 0,C 180,E1 9044.938,E2 9044.938} C_VEL
LIN {X 0,Y 606.409,Z 994.205,A -85,B 0,C 180,E1 9047.592,E2 9047.592} C_VEL
LIN {X 0,Y 596.262,Z 1063.375,A -85,B 0,C 180,E1 9051.699,E2 9051.699} C_VEL
LIN {X 0,Y 586.076,Z 1125.78,A -85,B 0,C 180,E1 9057.203,E2 9057.203} C_VEL
LIN {X 0,Y 578.006,Z 1177.28,A -85,B 0,C 180,E1 9063.748,E2 9063.748} C_VEL
LIN {X 0,Y 573.363,Z 1215.023,A -85,B 0,C 180,E1 9070.672,E2 9070.672} C_VEL
LIN {X 0,Y 571.389,Z 1239.236,A -85,B 0,C 180,E1 9077.338,E2 9077.338} C_VEL
LIN {X 0,Y 571.014,Z 1251.781,A -85,B 0,C 180,E1 9083.128,E2 9083.128} C_VEL
LIN {X 0,Y 570.696,Z 1256.847,A -85,B 0,C 180,E1 9089.237,E2 9089.237} C_VEL
LIN {X 0,Y 571.014,Z 1252.81,A -85,B 0,C 180,E1 9096.104,E2 9096.104} C_VEL
LIN {X 0,Y 572.155,Z 1235.511,A -85,B 0,C 180,E1 9103.815,E2 9103.815} C_VEL
LIN {X 0,Y 575.256,Z 1203.247,A -85,B 0,C 180,E1 9111.682,E2 9111.682} C_VEL
LIN {X 0,Y 581.469,Z 1156.892,A -85,B 0,C 180,E1 9119.036,E2 9119.036} C_VEL
LIN {X 0,Y 590.673,Z 1098.918,A -85,B 0,C 180,E1 9125.329,E2 9125.329} C_VEL
LIN {X 0,Y 600.805,Z 1033.057,A -85,B 0,C 180,E1 9130.241,E2 9130.241} C_VEL
LIN {X 0,Y 610.256,Z 959.672,A -85,B 0,C 180,E1 9133.805,E2 9133.805} C_VEL
LIN {X 0,Y 613.234,Z 915.548,A -85,B 0,C 180,E1 9135.274,E2 9135.274} C_VEL
LIN {X 0,Y 584.336,Z 862.646,A -85,B 0,C 180,E1 9139.704,E2 9139.704} C_VEL
LIN {X 0,Y 570.039,Z 839.06,A -85,B 0,C 180,E1 9142.037,E2 9142.037} C_VEL
LIN {X 0,Y 570.151,Z 839.06,A -85,B 0,C 180,E1 9150.559,E2 9150.559} C_VEL
LIN {X 0,Y 570.265,Z 839.06,A -85,B 0,C 180,E1 9158.998,E2 9158.998} C_VEL
LIN {X 0,Y 570.807,Z 839.06,A -85,B 0,C 180,E1 9168.546,E2 9168.546} C_VEL
LIN {X 0,Y 571.46,Z 839.06,A -85,B 0,C 180,E1 9179.283,E2 9179.283} C_VEL
LIN {X 0,Y 570.529,Z 839.06,A -85,B 0,C 180,E1 9188.454,E2 9188.454} C_VEL
LIN {X 0,Y 570.307,Z 839.06,A -85,B 0,C 180,E1 9196.266,E2 9196.266} C_VEL
LIN {X 0,Y 570.208,Z 839.06,A -85,B 0,C 180,E1 9204.405,E2 9204.405} C_VEL
LIN {X 0,Y 570.002,Z 839.06,A -85,B 0,C 180,E1 9213.122,E2 9213.122} C_VEL
LIN {X 0,Y 570.132,Z 840.365,A -85,B 0,C 180,E1 9217.614,E2 9217.614} C_VEL
LIN {X 0,Y 611.863,Z 909.016,A -85,B 0,C 180,E1 9223.597,E2 9223.597} C_VEL
LIN {X 0,Y 615.742,Z 921.211,A -85,B 0,C 180,E1 9224.265,E2 9224.265} C_VEL
LIN {X 0,Y 608.707,Z 1001.358,A -85,B 0,C 180,E1 9226.639,E2 9226.639} C_VEL
LIN {X 0,Y 599.208,Z 1074.248,A -85,B 0,C 180,E1 9230.432,E2 9230.432} C_VEL
LIN {X 0,Y 588.037,Z 1103.641,A -85,B 0,C 180,E1 9232.019,E2 9232.019} C_VEL
LIN {X 0,Y 577.615,Z 1165.135,A -85,B 0,C 180,E1 9237.845,E2 9237.845} C_VEL
LIN {X 0,Y 569.547,Z 1216.104,A -85,B 0,C 180,E1 9244.858,E2 9244.858} C_VEL
LIN {X 0,Y 564.955,Z 1253.068,A -85,B 0,C 180,E1 9252.382,E2 9252.382} C_VEL
LIN {X 0,Y 563.193,Z 1276.006,A -85,B 0,C 180,E1 9259.91,E2 9259.91} C_VEL
LIN {X 0,Y 562.9,Z 1285.349,A -85,B 0,C 180,E1 9266.134,E2 9266.134} C_VEL
LIN {X 0,Y 562.844,Z 1286.379,A -85,B 0,C 180,E1 9272.319,E2 9272.319} C_VEL
LIN {X 0,Y 563.345,Z 1277.589,A -85,B 0,C 180,E1 9279.305,E2 9279.305} C_VEL
LIN {X 0,Y 565.226,Z 1254.457,A -85,B 0,C 180,E1 9287.245,E2 9287.245} C_VEL
LIN {X 0,Y 569.66,Z 1215.774,A -85,B 0,C 180,E1 9295.194,E2 9295.194} C_VEL
LIN {X 0,Y 577.626,Z 1165.126,A -85,B 0,C 180,E1 9302.155,E2 9302.155} C_VEL
LIN {X 0,Y 588.094,Z 1103.654,A -85,B 0,C 180,E1 9307.976,E2 9307.976} C_VEL
LIN {X 0,Y 598.488,Z 1034.729,A -85,B 0,C 180,E1 9312.361,E2 9312.361} C_VEL
LIN {X 0,Y 607.284,Z 958.14,A -85,B 0,C 180,E1 9315.38,E2 9315.38} C_VEL
LIN {X 0,Y 609.275,Z 918.787,A -85,B 0,C 180,E1 9316.417,E2 9316.417} C_VEL
LIN {X 0,Y 573.514,Z 857.763,A -85,B 0,C 180,E1 9321.615,E2 9321.615} C_VEL
LIN {X 0,Y 562.142,Z 839.06,A -85,B 0,C 180,E1 9323.712,E2 9323.712} C_VEL
LIN {X 0,Y 562.368,Z 839.06,A -85,B 0,C 180,E1 9331.777,E2 9331.777} C_VEL
LIN {X 0,Y 562.022,Z 839.06,A -85,B 0,C 180,E1 9340.232,E2 9340.232} C_VEL
LIN {X 0,Y 562.622,Z 839.06,A -85,B 0,C 180,E1 9349.86,E2 9349.86} C_VEL
LIN {X 0,Y 563.478,Z 839.06,A -85,B 0,C 180,E1 9359.184,E2 9359.184} C_VEL
LIN {X 0,Y 562.627,Z 839.06,A -85,B 0,C 180,E1 9368.484,E2 9368.484} C_VEL
LIN {X 0,Y 562.246,Z 839.06,A -85,B 0,C 180,E1 9376.556,E2 9376.556} C_VEL
LIN {X 0,Y 562.135,Z 839.06,A -85,B 0,C 180,E1 9385.215,E2 9385.215} C_VEL
LIN {X 0,Y 561.919,Z 839.06,A -85,B 0,C 180,E1 9394.511,E2 9394.511} C_VEL
LIN {X 0,Y 562.187,Z 840.752,A -85,B 0,C 180,E1 9396.978,E2 9396.978} C_VEL
LIN {X 0,Y 600.958,Z 904.306,A -85,B 0,C 180,E1 9403.043,E2 9403.043} C_VEL
LIN {X 0,Y 608.177,Z 925.418,A -85,B 0,C 180,E1 9404.478,E2 9404.478} C_VEL
LIN {X 0,Y 600.091,Z 997.073,A -85,B 0,C 180,E1 9407.191,E2 9407.191} C_VEL
LIN {X 0,Y 589.498,Z 1065.089,A -85,B 0,C 180,E1 9411.324,E2 9411.324} C_VEL
LIN {X 0,Y 578.79,Z 1127.284,A -85,B 0,C 180,E1 9416.913,E2 9416.913} C_VEL
LIN {X 0,Y 570.257,Z 1178.981,A -85,B 0,C 180,E1 9423.637,E2 9423.637} C_VEL
LIN {X 0,Y 565.376,Z 1216.76,A -85,B 0,C 180,E1 9430.796,E2 9430.796} C_VEL
LIN {X 0,Y 563.395,Z 1240.381,A -85,B 0,C 180,E1 9437.551,E2 9437.551} C_VEL
LIN {X 0,Y 563.087,Z 1253.829,A -85,B 0,C 180,E1 9444.585,E2 9444.585} C_VEL
LIN {X 0,Y 563.302,Z 1256.35,A -85,B 0,C 180,E1 9452.316,E2 9452.316} C_VEL
LIN {X 0,Y 563.256,Z 1245.91,A -85,B 0,C 180,E1 9460.089,E2 9460.089} C_VEL
LIN {X 0,Y 564.669,Z 1223.99,A -85,B 0,C 180,E1 9467.34,E2 9467.34} C_VEL
LIN {X 0,Y 568.654,Z 1190.087,A -85,B 0,C 180,E1 9474.443,E2 9474.443} C_VEL
LIN {X 0,Y 576.197,Z 1142.722,A -85,B 0,C 180,E1 9481.24,E2 9481.24} C_VEL
LIN {X 0,Y 586.522,Z 1082.601,A -85,B 0,C 180,E1 9487.223,E2 9487.223} C_VEL
LIN {X 0,Y 597.696,Z 1013.979,A -85,B 0,C 180,E1 9491.847,E2 9491.847} C_VEL
LIN {X 0,Y 606.707,Z 939.973,A -85,B 0,C 180,E1 9495.007,E2 9495.007} C_VEL
LIN {X 0,Y 607.358,Z 918.911,A -85,B 0,C 180,E1 9495.737,E2 9495.737} C_VEL
LIN {X 0,Y 579.347,Z 867.082,A -85,B 0,C 180,E1 9500.206,E2 9500.206} C_VEL
LIN {X 0,Y 562.01,Z 839.06,A -85,B 0,C 180,E1 9503.202,E2 9503.202} C_VEL
LIN {X 0,Y 562.111,Z 839.06,A -85,B 0,C 180,E1 9511.864,E2 9511.864} C_VEL
LIN {X 0,Y 562.162,Z 839.06,A -85,B 0,C 180,E1 9520.331,E2 9520.331} C_VEL
LIN {X 0,Y 562.935,Z 839.06,A -85,B 0,C 180,E1 9529.841,E2 9529.841} C_VEL
LIN {X 0,Y 563.446,Z 839.06,A -85,B 0,C 180,E1 9539.273,E2 9539.273} C_VEL
LIN {X 0,Y 562.492,Z 839.06,A -85,B 0,C 180,E1 9548.576,E2 9548.576} C_VEL
LIN {X 0,Y 562.26,Z 839.06,A -85,B 0,C 180,E1 9556.564,E2 9556.564} C_VEL
LIN {X 0,Y 562.113,Z 839.06,A -85,B 0,C 180,E1 9565.212,E2 9565.212} C_VEL
LIN {X 0,Y 561.927,Z 839.06,A -85,B 0,C 180,E1 9574.514,E2 9574.514} C_VEL
LIN {X 0,Y 562.187,Z 840.681,A -85,B 0,C 180,E1 9576.566,E2 9576.566} C_VEL
LIN {X 0,Y 604.932,Z 909.701,A -85,B 0,C 180,E1 9582.924,E2 9582.924} C_VEL
LIN {X 0,Y 609.919,Z 924.56,A -85,B 0,C 180,E1 9583.795,E2 9583.795} C_VEL
LIN {X 0,Y 602.451,Z 1003.775,A -85,B 0,C 180,E1 9586.212,E2 9586.212} C_VEL
LIN {X 0,Y 592.453,Z 1076.588,A -85,B 0,C 180,E1 9590.078,E2 9590.078} C_VEL
LIN {X 0,Y 588.037,Z 1103.641,A -85,B 0,C 180,E1 9592.019,E2 9592.019} C_VEL
LIN {X 0,Y 576.547,Z 1131.406,A -85,B 0,C 180,E1 9593.881,E2 9593.881} C_VEL
LIN {X 0,Y 566.128,Z 1189.374,A -85,B 0,C 180,E1 9600.421,E2 9600.421} C_VEL
LIN {X 0,Y 559.278,Z 1232.914,A -85,B 0,C 180,E1 9607.548,E2 9607.548} C_VEL
LIN {X 0,Y 556.141,Z 1263.139,A -85,B 0,C 180,E1 9614.97,E2 9614.97} C_VEL
LIN {X 0,Y 555.481,Z 1281.704,A -85,B 0,C 180,E1 9622.936,E2 9622.936} C_VEL
LIN {X 0,Y 555.026,Z 1286.837,A -85,B 0,C 180,E1 9630.784,E2 9630.784} C_VEL
LIN {X 0,Y 555.07,Z 1280.491,A -85,B 0,C 180,E1 9637.86,E2 9637.86} C_VEL
LIN {X 0,Y 556.283,Z 1261.797,A -85,B 0,C 180,E1 9645.432,E2 9645.432} C_VEL
LIN {X 0,Y 560.367,Z 1228.148,A -85,B 0,C 180,E1 9653.342,E2 9653.342} C_VEL
LIN {X 0,Y 567.981,Z 1180.414,A -85,B 0,C 180,E1 9660.735,E2 9660.735} C_VEL
LIN {X 0,Y 578.126,Z 1122.805,A -85,B 0,C 180,E1 9666.882,E2 9666.882} C_VEL
LIN {X 0,Y 589.398,Z 1055.303,A -85,B 0,C 180,E1 9671.751,E2 9671.751} C_VEL
LIN {X 0,Y 599.568,Z 980.089,A -85,B 0,C 180,E1 9675.2,E2 9675.2} C_VEL
LIN {X 0,Y 603.303,Z 921.674,A -85,B 0,C 180,E1 9676.932,E2 9676.932} C_VEL
LIN {X 0,Y 568.695,Z 862.586,A -85,B 0,C 180,E1 9682.13,E2 9682.13} C_VEL
LIN {X 0,Y 554.149,Z 839.06,A -85,B 0,C 180,E1 9684.88,E2 9684.88} C_VEL
LIN {X 0,Y 554.373,Z 839.06,A -85,B 0,C 180,E1 9693.105,E2 9693.105} C_VEL
LIN {X 0,Y 554.31,Z 839.06,A -85,B 0,C 180,E1 9703.251,E2 9703.251} C_VEL
LIN {X 0,Y 554.628,Z 839.06,A -85,B 0,C 180,E1 9712.884,E2 9712.884} C_VEL
LIN {X 0,Y 554.831,Z 839.06,A -85,B 0,C 180,E1 9720.738,E2 9720.738} C_VEL
LIN {X 0,Y 554.591,Z 839.06,A -85,B 0,C 180,E1 9728.608,E2 9728.608} C_VEL
LIN {X 0,Y 554.239,Z 839.06,A -85,B 0,C 180,E1 9736.657,E2 9736.657} C_VEL
LIN {X 0,Y 554.141,Z 839.06,A -85,B 0,C 180,E1 9745.061,E2 9745.061} C_VEL
LIN {X 0,Y 553.907,Z 839.06,A -85,B 0,C 180,E1 9754.106,E2 9754.106} C_VEL
LIN {X 0,Y 554.07,Z 840.492,A -85,B 0,C 180,E1 9755.834,E2 9755.834} C_VEL
LIN {X 0,Y 593.582,Z 904.407,A -85,B 0,C 180,E1 9762.269,E2 9762.269} C_VEL
LIN {X 0,Y 602.308,Z 928.047,A -85,B 0,C 180,E1 9764.001,E2 9764.001} C_VEL
LIN {X 0,Y 593.724,Z 1000.253,A -85,B 0,C 180,E1 9766.796,E2 9766.796} C_VEL
LIN {X 0,Y 582.53,Z 1068.409,A -85,B 0,C 180,E1 9771.049,E2 9771.049} C_VEL
LIN {X 0,Y 570.95,Z 1131.955,A -85,B 0,C 180,E1 9776.969,E2 9776.969} C_VEL
LIN {X 0,Y 562.175,Z 1182.858,A -85,B 0,C 180,E1 9783.883,E2 9783.883} C_VEL
LIN {X 0,Y 557.365,Z 1218.498,A -85,B 0,C 180,E1 9790.922,E2 9790.922} C_VEL
LIN {X 0,Y 555.369,Z 1242.336,A -85,B 0,C 180,E1 9798.169,E2 9798.169} C_VEL
LIN {X 0,Y 555.147,Z 1254.776,A -85,B 0,C 180,E1 9805.373,E2 9805.373} C_VEL
LIN {X 0,Y 555.292,Z 1256.35,A -85,B 0,C 180,E1 9812.35,E2 9812.35} C_VEL
LIN {X 0,Y 555.278,Z 1245.912,A -85,B 0,C 180,E1 9820.236,E2 9820.236} C_VEL
LIN {X 0,Y 556.754,Z 1224.326,A -85,B 0,C 180,E1 9827.505,E2 9827.505} C_VEL
LIN {X 0,Y 561.04,Z 1190.089,A -85,B 0,C 180,E1 9834.797,E2 9834.797} C_VEL
LIN {X 0,Y 569.18,Z 1141.619,A -85,B 0,C 180,E1 9841.811,E2 9841.811} C_VEL
LIN {X 0,Y 580.038,Z 1081.839,A -85,B 0,C 180,E1 9847.783,E2 9847.783} C_VEL
LIN {X 0,Y 591.607,Z 1014.521,A -85,B 0,C 180,E1 9852.361,E2 9852.361} C_VEL
LIN {X 0,Y 600.944,Z 941.467,A -85,B 0,C 180,E1 9855.512,E2 9855.512} C_VEL
LIN {X 0,Y 601.559,Z 922.186,A -85,B 0,C 180,E1 9856.207,E2 9856.207} C_VEL
LIN {X 0,Y 573.095,Z 869.446,A -85,B 0,C 180,E1 9860.915,E2 9860.915} C_VEL
LIN {X 0,Y 553.965,Z 839.06,A -85,B 0,C 180,E1 9864.217,E2 9864.217} C_VEL
LIN {X 0,Y 554.078,Z 839.06,A -85,B 0,C 180,E1 9873.191,E2 9873.191} C_VEL
LIN {X 0,Y 554.152,Z 839.06,A -85,B 0,C 180,E1 9881.696,E2 9881.696} C_VEL
LIN {X 0,Y 554.948,Z 839.06,A -85,B 0,C 180,E1 9889.81,E2 9889.81} C_VEL
LIN {X 0,Y 555.432,Z 839.06,A -85,B 0,C 180,E1 9899.262,E2 9899.262} C_VEL
LIN {X 0,Y 554.461,Z 839.06,A -85,B 0,C 180,E1 9908.701,E2 9908.701} C_VEL
LIN {X 0,Y 554.243,Z 839.06,A -85,B 0,C 180,E1 9916.751,E2 9916.751} C_VEL
LIN {X 0,Y 554.13,Z 839.06,A -85,B 0,C 180,E1 9925.161,E2 9925.161} C_VEL
LIN {X 0,Y 553.913,Z 839.06,A -85,B 0,C 180,E1 9934.214,E2 9934.214} C_VEL
LIN {X 0,Y 554.215,Z 840.9,A -85,B 0,C 180,E1 9935.455,E2 9935.455} C_VEL
LIN {X 0,Y 595.912,Z 906.864,A -85,B 0,C 180,E1 9941.933,E2 9941.933} C_VEL
LIN {X 0,Y 604.227,Z 926.584,A -85,B 0,C 180,E1 9943.29,E2 9943.29} C_VEL
LIN {X 0,Y 596.337,Z 1005.362,A -85,B 0,C 180,E1 9945.742,E2 9945.742} C_VEL
LIN {X 0,Y 585.654,Z 1079.167,A -85,B 0,C 180,E1 9949.743,E2 9949.743} C_VEL
LIN {X 0,Y 576.547,Z 1131.406,A -85,B 0,C 180,E1 9953.881,E2 9953.881} C_VEL
LIN {X 0,Y 565.029,Z 1157.232,A -85,B 0,C 180,E1 9956.039,E2 9956.039} C_VEL
LIN {X 0,Y 555.662,Z 1209.594,A -85,B 0,C 180,E1 9963.037,E2 9963.037} C_VEL
LIN {X 0,Y 549.924,Z 1250.046,A -85,B 0,C 180,E1 9971.073,E2 9971.073} C_VEL
LIN {X 0,Y 547.492,Z 1274.16,A -85,B 0,C 180,E1 9978.808,E2 9978.808} C_VEL
LIN {X 0,Y 546.916,Z 1285.349,A -85,B 0,C 180,E1 9986.021,E2 9986.021} C_VEL
LIN {X 0,Y 546.882,Z 1286.38,A -85,B 0,C 180,E1 9992.387,E2 9992.387} C_VEL
LIN {X 0,Y 547.637,Z 1276.431,A -85,B 0,C 180,E1 10000.167,E2 10000.167} C_VEL
LIN {X 0,Y 549.504,Z 1251.605,A -85,B 0,C 180,E1 10008.525,E2 10008.525} C_VEL
LIN {X 0,Y 554.81,Z 1213.101,A -85,B 0,C 180,E1 10016.401,E2 10016.401} C_VEL
LIN {X 0,Y 564.303,Z 1160.568,A -85,B 0,C 180,E1 10023.606,E2 10023.606} C_VEL
LIN {X 0,Y 575.75,Z 1099.172,A -85,B 0,C 180,E1 10029.336,E2 10029.336} C_VEL
LIN {X 0,Y 587.572,Z 1027.846,A -85,B 0,C 180,E1 10033.76,E2 10033.76} C_VEL
LIN {X 0,Y 596.733,Z 950.456,A -85,B 0,C 180,E1 10036.698,E2 10036.698} C_VEL
LIN {X 0,Y 597.631,Z 925.073,A -85,B 0,C 180,E1 10037.418,E2 10037.418} C_VEL
LIN {X 0,Y 562.295,Z 864.419,A -85,B 0,C 180,E1 10042.933,E2 10042.933} C_VEL
LIN {X 0,Y 546.162,Z 839.06,A -85,B 0,C 180,E1 10045.896,E2 10045.896} C_VEL
LIN {X 0,Y 546.32,Z 839.06,A -85,B 0,C 180,E1 10054.571,E2 10054.571} C_VEL
LIN {X 0,Y 546.289,Z 839.06,A -85,B 0,C 180,E1 10064.655,E2 10064.655} C_VEL
LIN {X 0,Y 546.625,Z 839.06,A -85,B 0,C 180,E1 10072.779,E2 10072.779} C_VEL
LIN {X 0,Y 546.829,Z 839.06,A -85,B 0,C 180,E1 10080.749,E2 10080.749} C_VEL
LIN {X 0,Y 546.429,Z 839.06,A -85,B 0,C 180,E1 10089.499,E2 10089.499} C_VEL
LIN {X 0,Y 546.051,Z 839.06,A -85,B 0,C 180,E1 10098.586,E2 10098.586} C_VEL
LIN {X 0,Y 546.069,Z 839.06,A -85,B 0,C 180,E1 10107.235,E2 10107.235} C_VEL
LIN {X 0,Y 546.114,Z 840.885,A -85,B 0,C 180,E1 10114.661,E2 10114.661} C_VEL
LIN {X 0,Y 585.081,Z 902.426,A -85,B 0,C 180,E1 10121.276,E2 10121.276} C_VEL
LIN {X 0,Y 596.381,Z 931.47,A -85,B 0,C 180,E1 10123.537,E2 10123.537} C_VEL
LIN {X 0,Y 587.363,Z 1003.55,A -85,B 0,C 180,E1 10126.416,E2 10126.416} C_VEL
LIN {X 0,Y 575.807,Z 1070.38,A -85,B 0,C 180,E1 10130.667,E2 10130.667} C_VEL
LIN {X 0,Y 563.586,Z 1133.705,A -85,B 0,C 180,E1 10136.712,E2 10136.712} C_VEL
LIN {X 0,Y 554.409,Z 1184.398,A -85,B 0,C 180,E1 10143.769,E2 10143.769} C_VEL
LIN {X 0,Y 549.378,Z 1220.214,A -85,B 0,C 180,E1 10151.053,E2 10151.053} C_VEL
LIN {X 0,Y 547.389,Z 1243.357,A -85,B 0,C 180,E1 10158.424,E2 10158.424} C_VEL
LIN {X 0,Y 547.278,Z 1255.378,A -85,B 0,C 180,E1 10166.023,E2 10166.023} C_VEL
LIN {X 0,Y 547.089,Z 1255.319,A -85,B 0,C 180,E1 10173.977,E2 10173.977} C_VEL
LIN {X 0,Y 547.297,Z 1244.055,A -85,B 0,C 180,E1 10181.195,E2 10181.195} C_VEL
LIN {X 0,Y 549.002,Z 1223.318,A -85,B 0,C 180,E1 10188.034,E2 10188.034} C_VEL
LIN {X 0,Y 553.682,Z 1188.793,A -85,B 0,C 180,E1 10195.383,E2 10195.383} C_VEL
LIN {X 0,Y 562.39,Z 1140.054,A -85,B 0,C 180,E1 10202.446,E2 10202.446} C_VEL
LIN {X 0,Y 574.497,Z 1077.178,A -85,B 0,C 180,E1 10208.687,E2 10208.687} C_VEL
LIN {X 0,Y 586.306,Z 1010.412,A -85,B 0,C 180,E1 10213.129,E2 10213.129} C_VEL
LIN {X 0,Y 595.748,Z 938.267,A -85,B 0,C 180,E1 10216.163,E2 10216.163} C_VEL
LIN {X 0,Y 595.319,Z 924.497,A -85,B 0,C 180,E1 10216.767,E2 10216.767} C_VEL
LIN {X 0,Y 565.949,Z 870.216,A -85,B 0,C 180,E1 10221.806,E2 10221.806} C_VEL
LIN {X 0,Y 545.928,Z 839.06,A -85,B 0,C 180,E1 10225.325,E2 10225.325} C_VEL
LIN {X 0,Y 546.105,Z 839.06,A -85,B 0,C 180,E1 10234.617,E2 10234.617} C_VEL
LIN {X 0,Y 546.521,Z 839.06,A -85,B 0,C 180,E1 10244.756,E2 10244.756} C_VEL
LIN {X 0,Y 546.636,Z 839.06,A -85,B 0,C 180,E1 10252.871,E2 10252.871} C_VEL
LIN {X 0,Y 546.753,Z 839.06,A -85,B 0,C 180,E1 10260.841,E2 10260.841} C_VEL
LIN {X 0,Y 546.326,Z 839.06,A -85,B 0,C 180,E1 10269.44,E2 10269.44} C_VEL
LIN {X 0,Y 546.069,Z 839.06,A -85,B 0,C 180,E1 10278.682,E2 10278.682} C_VEL
LIN {X 0,Y 546.031,Z 839.06,A -85,B 0,C 180,E1 10287.34,E2 10287.34} C_VEL
LIN {X 0,Y 546.071,Z 840.599,A -85,B 0,C 180,E1 10294.242,E2 10294.242} C_VEL
LIN {X 0,Y 587.034,Z 904.378,A -85,B 0,C 180,E1 10300.915,E2 10300.915} C_VEL
LIN {X 0,Y 598.491,Z 930.186,A -85,B 0,C 180,E1 10302.808,E2 10302.808} C_VEL
LIN {X 0,Y 589.843,Z 1010.166,A -85,B 0,C 180,E1 10305.4,E2 10305.4} C_VEL
LIN {X 0,Y 578.502,Z 1083.605,A -85,B 0,C 180,E1 10309.532,E2 10309.532} C_VEL
LIN {X 0,Y 567.086,Z 1146.33,A -85,B 0,C 180,E1 10314.861,E2 10314.861} C_VEL
LIN {X 0,Y 565.029,Z 1157.232,A -85,B 0,C 180,E1 10316.039,E2 10316.039} C_VEL
LIN {X 0,Y 553.142,Z 1181.112,A -85,B 0,C 180,E1 10318.448,E2 10318.448} C_VEL
LIN {X 0,Y 544.852,Z 1227.347,A -85,B 0,C 180,E1 10325.791,E2 10325.791} C_VEL
LIN {X 0,Y 540.603,Z 1259.113,A -85,B 0,C 180,E1 10333.272,E2 10333.272} C_VEL
LIN {X 0,Y 539.21,Z 1277.268,A -85,B 0,C 180,E1 10340.111,E2 10340.111} C_VEL
LIN {X 0,Y 539.143,Z 1286.38,A -85,B 0,C 180,E1 10347.58,E2 10347.58} C_VEL
LIN {X 0,Y 539.344,Z 1283.771,A -85,B 0,C 180,E1 10355.654,E2 10355.654} C_VEL
LIN {X 0,Y 539.714,Z 1269.101,A -85,B 0,C 180,E1 10363.419,E2 10363.419} C_VEL
LIN {X 0,Y 542.213,Z 1244.822,A -85,B 0,C 180,E1 10370.487,E2 10370.487} C_VEL
LIN {X 0,Y 548.27,Z 1207.176,A -85,B 0,C 180,E1 10377.763,E2 10377.763} C_VEL
LIN {X 0,Y 558.469,Z 1154.395,A -85,B 0,C 180,E1 10384.764,E2 10384.764} C_VEL
LIN {X 0,Y 570.96,Z 1089.974,A -85,B 0,C 180,E1 10390.525,E2 10390.525} C_VEL
LIN {X 0,Y 582.893,Z 1019.629,A -85,B 0,C 180,E1 10394.684,E2 10394.684} C_VEL
LIN {X 0,Y 591.959,Z 942.893,A -85,B 0,C 180,E1 10397.44,E2 10397.44} C_VEL
LIN {X 0,Y 591.645,Z 927.704,A -85,B 0,C 180,E1 10397.972,E2 10397.972} C_VEL
LIN {X 0,Y 556.556,Z 867.658,A -85,B 0,C 180,E1 10403.647,E2 10403.647} C_VEL
LIN {X 0,Y 538.169,Z 839.06,A -85,B 0,C 180,E1 10407.224,E2 10407.224} C_VEL
LIN {X 0,Y 538.139,Z 839.06,A -85,B 0,C 180,E1 10416.47,E2 10416.47} C_VEL
LIN {X 0,Y 538.292,Z 839.06,A -85,B 0,C 180,E1 10426.654,E2 10426.654} C_VEL
LIN {X 0,Y 538.448,Z 839.06,A -85,B 0,C 180,E1 10434.294,E2 10434.294} C_VEL
LIN {X 0,Y 538.827,Z 839.06,A -85,B 0,C 180,E1 10440.76,E2 10440.76} C_VEL
LIN {X 0,Y 538.555,Z 839.06,A -85,B 0,C 180,E1 10448.867,E2 10448.867} C_VEL
LIN {X 0,Y 538.131,Z 839.06,A -85,B 0,C 180,E1 10457.171,E2 10457.171} C_VEL
LIN {X 0,Y 538.051,Z 839.06,A -85,B 0,C 180,E1 10465.865,E2 10465.865} C_VEL
LIN {X 0,Y 538.017,Z 840.295,A -85,B 0,C 180,E1 10473.369,E2 10473.369} C_VEL
LIN {X 0,Y 576.656,Z 900.996,A -85,B 0,C 180,E1 10480.259,E2 10480.259} C_VEL
LIN {X 0,Y 590.612,Z 934.013,A -85,B 0,C 180,E1 10483.039,E2 10483.039} C_VEL
LIN {X 0,Y 581.097,Z 1006.125,A -85,B 0,C 180,E1 10485.985,E2 10485.985} C_VEL
LIN {X 0,Y 569.211,Z 1071.864,A -85,B 0,C 180,E1 10490.243,E2 10490.243} C_VEL
LIN {X 0,Y 556.521,Z 1134.086,A -85,B 0,C 180,E1 10496.285,E2 10496.285} C_VEL
LIN {X 0,Y 546.884,Z 1184.552,A -85,B 0,C 180,E1 10503.409,E2 10503.409} C_VEL
LIN {X 0,Y 541.554,Z 1220.212,A -85,B 0,C 180,E1 10510.768,E2 10510.768} C_VEL
LIN {X 0,Y 539.432,Z 1242.332,A -85,B 0,C 180,E1 10517.814,E2 10517.814} C_VEL
LIN {X 0,Y 539.08,Z 1253.819,A -85,B 0,C 180,E1 10524.343,E2 10524.343} C_VEL
LIN {X 0,Y 539.291,Z 1256.351,A -85,B 0,C 180,E1 10532.42,E2 10532.42} C_VEL
LIN {X 0,Y 539.38,Z 1247.565,A -85,B 0,C 180,E1 10539.686,E2 10539.686} C_VEL
LIN {X 0,Y 540.787,Z 1227.594,A -85,B 0,C 180,E1 10547.143,E2 10547.143} C_VEL
LIN {X 0,Y 545.194,Z 1194.687,A -85,B 0,C 180,E1 10554.684,E2 10554.684} C_VEL
LIN {X 0,Y 553.919,Z 1147.199,A -85,B 0,C 180,E1 10562.021,E2 10562.021} C_VEL
LIN {X 0,Y 566.557,Z 1085.217,A -85,B 0,C 180,E1 10568.568,E2 10568.568} C_VEL
LIN {X 0,Y 579.33,Z 1017.435,A -85,B 0,C 180,E1 10573.317,E2 10573.317} C_VEL
LIN {X 0,Y 589.639,Z 943.544,A -85,B 0,C 180,E1 10576.579,E2 10576.579} C_VEL
LIN {X 0,Y 589.571,Z 928,A -85,B 0,C 180,E1 10577.231,E2 10577.231} C_VEL
LIN {X 0,Y 561.564,Z 875.593,A -85,B 0,C 180,E1 10582.253,E2 10582.253} C_VEL
LIN {X 0,Y 537.874,Z 839.06,A -85,B 0,C 180,E1 10586.686,E2 10586.686} C_VEL
LIN {X 0,Y 538.186,Z 839.06,A -85,B 0,C 180,E1 10596.456,E2 10596.456} C_VEL
LIN {X 0,Y 538.673,Z 839.06,A -85,B 0,C 180,E1 10606.48,E2 10606.48} C_VEL
LIN {X 0,Y 538.438,Z 839.06,A -85,B 0,C 180,E1 10614.387,E2 10614.387} C_VEL
LIN {X 0,Y 538.768,Z 839.06,A -85,B 0,C 180,E1 10620.853,E2 10620.853} C_VEL
LIN {X 0,Y 538.414,Z 839.06,A -85,B 0,C 180,E1 10628.963,E2 10628.963} C_VEL
LIN {X 0,Y 538.149,Z 839.06,A -85,B 0,C 180,E1 10637.267,E2 10637.267} C_VEL
LIN {X 0,Y 538.036,Z 839.06,A -85,B 0,C 180,E1 10645.969,E2 10645.969} C_VEL
LIN {X 0,Y 538.005,Z 840.373,A -85,B 0,C 180,E1 10652.966,E2 10652.966} C_VEL
LIN {X 0,Y 579.073,Z 903.618,A -85,B 0,C 180,E1 10659.99,E2 10659.99} C_VEL
LIN {X 0,Y 592.715,Z 933.922,A -85,B 0,C 180,E1 10662.333,E2 10662.333} C_VEL
LIN {X 0,Y 583.741,Z 1011.716,A -85,B 0,C 180,E1 10664.918,E2 10664.918} C_VEL
LIN {X 0,Y 571.895,Z 1084.799,A -85,B 0,C 180,E1 10669.096,E2 10669.096} C_VEL
LIN {X 0,Y 559.589,Z 1149.469,A -85,B 0,C 180,E1 10674.709,E2 10674.709} C_VEL
LIN {X 0,Y 553.142,Z 1181.112,A -85,B 0,C 180,E1 10678.448,E2 10678.448} C_VEL
LIN {X 0,Y 541.867,Z 1202.849,A -85,B 0,C 180,E1 10681.137,E2 10681.137} C_VEL
LIN {X 0,Y 534.88,Z 1244.829,A -85,B 0,C 180,E1 10689.221,E2 10689.221} C_VEL
LIN {X 0,Y 531.944,Z 1272.229,A -85,B 0,C 180,E1 10697.641,E2 10697.641} C_VEL
LIN {X 0,Y 531.246,Z 1283.768,A -85,B 0,C 180,E1 10704.26,E2 10704.26} C_VEL
LIN {X 0,Y 531.047,Z 1286.837,A -85,B 0,C 180,E1 10710.819,E2 10710.819} C_VEL
LIN {X 0,Y 531.133,Z 1280.482,A -85,B 0,C 180,E1 10718.217,E2 10718.217} C_VEL
LIN {X 0,Y 532.743,Z 1261.794,A -85,B 0,C 180,E1 10726.132,E2 10726.132} C_VEL
LIN {X 0,Y 537.805,Z 1227.397,A -85,B 0,C 180,E1 10734.536,E2 10734.536} C_VEL
LIN {X 0,Y 546.529,Z 1179.889,A -85,B 0,C 180,E1 10742.158,E2 10742.158} C_VEL
LIN {X 0,Y 558.469,Z 1120.886,A -85,B 0,C 180,E1 10748.547,E2 10748.547} C_VEL
LIN {X 0,Y 571.53,Z 1051.355,A -85,B 0,C 180,E1 10753.608,E2 10753.608} C_VEL
LIN {X 0,Y 583.059,Z 975.284,A -85,B 0,C 180,E1 10757.051,E2 10757.051} C_VEL
LIN {X 0,Y 586.32,Z 931.791,A -85,B 0,C 180,E1 10758.421,E2 10758.421} C_VEL
LIN {X 0,Y 551.531,Z 871.413,A -85,B 0,C 180,E1 10764.275,E2 10764.275} C_VEL
LIN {X 0,Y 530.195,Z 839.06,A -85,B 0,C 180,E1 10768.412,E2 10768.412} C_VEL
LIN {X 0,Y 530.05,Z 839.06,A -85,B 0,C 180,E1 10777.217,E2 10777.217} C_VEL
LIN {X 0,Y 530.264,Z 839.06,A -85,B 0,C 180,E1 10785.876,E2 10785.876} C_VEL
LIN {X 0,Y 530.449,Z 839.06,A -85,B 0,C 180,E1 10794.207,E2 10794.207} C_VEL
LIN {X 0,Y 530.819,Z 839.06,A -85,B 0,C 180,E1 10800.772,E2 10800.772} C_VEL
LIN {X 0,Y 530.5,Z 839.06,A -85,B 0,C 180,E1 10809.147,E2 10809.147} C_VEL
LIN {X 0,Y 530.095,Z 839.06,A -85,B 0,C 180,E1 10817.44,E2 10817.44} C_VEL
LIN {X 0,Y 530.054,Z 839.06,A -85,B 0,C 180,E1 10826.285,E2 10826.285} C_VEL
LIN {X 0,Y 530.169,Z 841.078,A -85,B 0,C 180,E1 10832.068,E2 10832.068} C_VEL
LIN {X 0,Y 566.317,Z 896.075,A -85,B 0,C 180,E1 10838.839,E2 10838.839} C_VEL
LIN {X 0,Y 585.038,Z 935.408,A -85,B 0,C 180,E1 10842.5,E2 10842.5} C_VEL
LIN {X 0,Y 575.015,Z 1007.842,A -85,B 0,C 180,E1 10845.499,E2 10845.499} C_VEL
LIN {X 0,Y 562.45,Z 1074.219,A -85,B 0,C 180,E1 10849.879,E2 10849.879} C_VEL
LIN {X 0,Y 549.266,Z 1135.629,A -85,B 0,C 180,E1 10855.981,E2 10855.981} C_VEL
LIN {X 0,Y 539.17,Z 1185.747,A -85,B 0,C 180,E1 10863.223,E2 10863.223} C_VEL
LIN {X 0,Y 533.747,Z 1220.268,A -85,B 0,C 180,E1 10870.491,E2 10870.491} C_VEL
LIN {X 0,Y 531.461,Z 1242.33,A -85,B 0,C 180,E1 10877.629,E2 10877.629} C_VEL
LIN {X 0,Y 531.071,Z 1253.815,A -85,B 0,C 180,E1 10884.257,E2 10884.257} C_VEL
LIN {X 0,Y 531.288,Z 1256.352,A -85,B 0,C 180,E1 10892.456,E2 10892.456} C_VEL
LIN {X 0,Y 531.331,Z 1246.942,A -85,B 0,C 180,E1 10900.163,E2 10900.163} C_VEL
LIN {X 0,Y 533.059,Z 1225.708,A -85,B 0,C 180,E1 10907.925,E2 10907.925} C_VEL
LIN {X 0,Y 537.936,Z 1192.665,A -85,B 0,C 180,E1 10915.453,E2 10915.453} C_VEL
LIN {X 0,Y 547.575,Z 1143.791,A -85,B 0,C 180,E1 10922.933,E2 10922.933} C_VEL
LIN {X 0,Y 560.588,Z 1083.333,A -85,B 0,C 180,E1 10929.272,E2 10929.272} C_VEL
LIN {X 0,Y 573.543,Z 1016.855,A -85,B 0,C 180,E1 10933.924,E2 10933.924} C_VEL
LIN {X 0,Y 584.225,Z 943.244,A -85,B 0,C 180,E1 10937.168,E2 10937.168} C_VEL
LIN {X 0,Y 583.736,Z 931.162,A -85,B 0,C 180,E1 10937.732,E2 10937.732} C_VEL
LIN {X 0,Y 554.84,Z 876.974,A -85,B 0,C 180,E1 10943.134,E2 10943.134} C_VEL
LIN {X 0,Y 529.904,Z 839.06,A -85,B 0,C 180,E1 10948.072,E2 10948.072} C_VEL
LIN {X 0,Y 530.145,Z 839.06,A -85,B 0,C 180,E1 10957.324,E2 10957.324} C_VEL
LIN {X 0,Y 530.687,Z 839.06,A -85,B 0,C 180,E1 10967.667,E2 10967.667} C_VEL
LIN {X 0,Y 530.855,Z 839.06,A -85,B 0,C 180,E1 10977.59,E2 10977.59} C_VEL
LIN {X 0,Y 530.699,Z 839.06,A -85,B 0,C 180,E1 10987.439,E2 10987.439} C_VEL
LIN {X 0,Y 530.109,Z 839.06,A -85,B 0,C 180,E1 10997.538,E2 10997.538} C_VEL
LIN {X 0,Y 530.023,Z 839.06,A -85,B 0,C 180,E1 11006.392,E2 11006.392} C_VEL
LIN {X 0,Y 530.19,Z 841.106,A -85,B 0,C 180,E1 11011.671,E2 11011.671} C_VEL
LIN {X 0,Y 567.209,Z 896.555,A -85,B 0,C 180,E1 11018.389,E2 11018.389} C_VEL
LIN {X 0,Y 587.05,Z 936.438,A -85,B 0,C 180,E1 11021.82,E2 11021.82} C_VEL
LIN {X 0,Y 577.449,Z 1014.854,A -85,B 0,C 180,E1 11024.501,E2 11024.501} C_VEL
LIN {X 0,Y 565.258,Z 1086.384,A -85,B 0,C 180,E1 11028.68,E2 11028.68} C_VEL
LIN {X 0,Y 552.549,Z 1150.005,A -85,B 0,C 180,E1 11034.291,E2 11034.291} C_VEL
LIN {X 0,Y 541.867,Z 1202.849,A -85,B 0,C 180,E1 11041.137,E2 11041.137} C_VEL
LIN {X 0,Y 530.774,Z 1222.434,A -85,B 0,C 180,E1 11044.087,E2 11044.087} C_VEL
LIN {X 0,Y 525.14,Z 1257.751,A -85,B 0,C 180,E1 11052.33,E2 11052.33} C_VEL
LIN {X 0,Y 523.294,Z 1277.108,A -85,B 0,C 180,E1 11059.724,E2 11059.724} C_VEL
LIN {X 0,Y 522.962,Z 1285.348,A -85,B 0,C 180,E1 11065.839,E2 11065.839} C_VEL
LIN {X 0,Y 522.915,Z 1286.38,A -85,B 0,C 180,E1 11072.496,E2 11072.496} C_VEL
LIN {X 0,Y 523.527,Z 1277.859,A -85,B 0,C 180,E1 11079.867,E2 11079.867} C_VEL
LIN {X 0,Y 525.699,Z 1254.681,A -85,B 0,C 180,E1 11088.522,E2 11088.522} C_VEL
LIN {X 0,Y 531.495,Z 1217.983,A -85,B 0,C 180,E1 11096.723,E2 11096.723} C_VEL
LIN {X 0,Y 541.687,Z 1168.34,A -85,B 0,C 180,E1 11104.095,E2 11104.095} C_VEL
LIN {X 0,Y 555.008,Z 1105.961,A -85,B 0,C 180,E1 11110.346,E2 11110.346} C_VEL
LIN {X 0,Y 568.493,Z 1035.322,A -85,B 0,C 180,E1 11115.046,E2 11115.046} C_VEL
LIN {X 0,Y 579.418,Z 957.666,A -85,B 0,C 180,E1 11118.21,E2 11118.21} C_VEL
LIN {X 0,Y 580.41,Z 934.575,A -85,B 0,C 180,E1 11118.974,E2 11118.974} C_VEL
LIN {X 0,Y 546.521,Z 875.632,A -85,B 0,C 180,E1 11124.912,E2 11124.912} C_VEL
LIN {X 0,Y 522.23,Z 839.06,A -85,B 0,C 180,E1 11129.871,E2 11129.871} C_VEL
LIN {X 0,Y 521.963,Z 839.06,A -85,B 0,C 180,E1 11138.643,E2 11138.643} C_VEL
LIN {X 0,Y 522.258,Z 839.06,A -85,B 0,C 180,E1 11147.367,E2 11147.367} C_VEL
LIN {X 0,Y 522.489,Z 839.06,A -85,B 0,C 180,E1 11155.789,E2 11155.789} C_VEL
LIN {X 0,Y 522.499,Z 839.06,A -85,B 0,C 180,E1 11162.449,E2 11162.449} C_VEL
LIN {X 0,Y 522.308,Z 839.06,A -85,B 0,C 180,E1 11170.835,E2 11170.835} C_VEL
LIN {X 0,Y 522.005,Z 839.06,A -85,B 0,C 180,E1 11179.476,E2 11179.476} C_VEL
LIN {X 0,Y 521.954,Z 839.06,A -85,B 0,C 180,E1 11188.606,E2 11188.606} C_VEL
LIN {X 0,Y 522.141,Z 841.067,A -85,B 0,C 180,E1 11190.621,E2 11190.621} C_VEL
LIN {X 0,Y 557.613,Z 893.93,A -85,B 0,C 180,E1 11197.63,E2 11197.63} C_VEL
LIN {X 0,Y 579.229,Z 939.239,A -85,B 0,C 180,E1 11202.022,E2 11202.022} C_VEL
LIN {X 0,Y 568.516,Z 1012.171,A -85,B 0,C 180,E1 11205.143,E2 11205.143} C_VEL
LIN {X 0,Y 555.103,Z 1079.489,A -85,B 0,C 180,E1 11209.752,E2 11209.752} C_VEL
LIN {X 0,Y 541.592,Z 1139.488,A -85,B 0,C 180,E1 11215.936,E2 11215.936} C_VEL
LIN {X 0,Y 530.893,Z 1190.563,A -85,B 0,C 180,E1 11223.689,E2 11223.689} C_VEL
LIN {X 0,Y 525.353,Z 1226.563,A -85,B 0,C 180,E1 11231.954,E2 11231.954} C_VEL
LIN {X 0,Y 523.588,Z 1248.199,A -85,B 0,C 180,E1 11240.272,E2 11240.272} C_VEL
LIN {X 0,Y 523.063,Z 1256.408,A -85,B 0,C 180,E1 11247.504,E2 11247.504} C_VEL
LIN {X 0,Y 523.081,Z 1255.32,A -85,B 0,C 180,E1 11254.16,E2 11254.16} C_VEL
LIN {X 0,Y 523.43,Z 1244.057,A -85,B 0,C 180,E1 11261.713,E2 11261.713} C_VEL
LIN {X 0,Y 525.847,Z 1221.452,A -85,B 0,C 180,E1 11269.39,E2 11269.39} C_VEL
LIN {X 0,Y 532.489,Z 1182.868,A -85,B 0,C 180,E1 11277.599,E2 11277.599} C_VEL
LIN {X 0,Y 544.239,Z 1128.361,A -85,B 0,C 180,E1 11285.315,E2 11285.315} C_VEL
LIN {X 0,Y 557.767,Z 1067.052,A -85,B 0,C 180,E1 11291.172,E2 11291.172} C_VEL
LIN {X 0,Y 570.975,Z 998.506,A -85,B 0,C 180,E1 11295.478,E2 11295.478} C_VEL
LIN {X 0,Y 578.377,Z 935.484,A -85,B 0,C 180,E1 11298.144,E2 11298.144} C_VEL
LIN {X 0,Y 550.318,Z 882.018,A -85,B 0,C 180,E1 11303.643,E2 11303.643} C_VEL
LIN {X 0,Y 521.9,Z 839.06,A -85,B 0,C 180,E1 11309.476,E2 11309.476} C_VEL
LIN {X 0,Y 522.128,Z 839.06,A -85,B 0,C 180,E1 11318.753,E2 11318.753} C_VEL
LIN {X 0,Y 522.652,Z 839.06,A -85,B 0,C 180,E1 11327.474,E2 11327.474} C_VEL
LIN {X 0,Y 522.851,Z 839.06,A -85,B 0,C 180,E1 11337.553,E2 11337.553} C_VEL
LIN {X 0,Y 522.675,Z 839.06,A -85,B 0,C 180,E1 11347.554,E2 11347.554} C_VEL
LIN {X 0,Y 522.067,Z 839.06,A -85,B 0,C 180,E1 11357.817,E2 11357.817} C_VEL
LIN {X 0,Y 521.929,Z 839.06,A -85,B 0,C 180,E1 11367.485,E2 11367.485} C_VEL
LIN {X 0,Y 522.158,Z 841.034,A -85,B 0,C 180,E1 11370.225,E2 11370.225} C_VEL
LIN {X 0,Y 558.89,Z 895.075,A -85,B 0,C 180,E1 11377.275,E2 11377.275} C_VEL
LIN {X 0,Y 581.449,Z 938.785,A -85,B 0,C 180,E1 11381.293,E2 11381.293} C_VEL
LIN {X 0,Y 571.251,Z 1017.515,A -85,B 0,C 180,E1 11384.05,E2 11384.05} C_VEL
LIN {X 0,Y 558.35,Z 1089.33,A -85,B 0,C 180,E1 11388.352,E2 11388.352} C_VEL
LIN {X 0,Y 545.102,Z 1152.634,A -85,B 0,C 180,E1 11394.093,E2 11394.093} C_VEL
LIN {X 0,Y 534.069,Z 1205.293,A -85,B 0,C 180,E1 11401.104,E2 11401.104} C_VEL
LIN {X 0,Y 530.774,Z 1222.434,A -85,B 0,C 180,E1 11404.087,E2 11404.087} C_VEL
LIN {X 0,Y 519.868,Z 1239.481,A -85,B 0,C 180,E1 11407.271,E2 11407.271} C_VEL
LIN {X 0,Y 516.279,Z 1267.95,A -85,B 0,C 180,E1 11415.526,E2 11415.526} C_VEL
LIN {X 0,Y 515.285,Z 1283.762,A -85,B 0,C 180,E1 11424.082,E2 11424.082} C_VEL
LIN {X 0,Y 515.067,Z 1286.836,A -85,B 0,C 180,E1 11430.845,E2 11430.845} C_VEL
LIN {X 0,Y 515.176,Z 1280.563,A -85,B 0,C 180,E1 11438.412,E2 11438.412} C_VEL
LIN {X 0,Y 517.182,Z 1261.089,A -85,B 0,C 180,E1 11446.861,E2 11446.861} C_VEL
LIN {X 0,Y 522.623,Z 1226.761,A -85,B 0,C 180,E1 11455.431,E2 11455.431} C_VEL
LIN {X 0,Y 531.954,Z 1181.332,A -85,B 0,C 180,E1 11462.881,E2 11462.881} C_VEL
LIN {X 0,Y 545.237,Z 1121.235,A -85,B 0,C 180,E1 11469.564,E2 11469.564} C_VEL
LIN {X 0,Y 559.461,Z 1052.012,A -85,B 0,C 180,E1 11474.702,E2 11474.702} C_VEL
LIN {X 0,Y 571.83,Z 976.613,A -85,B 0,C 180,E1 11478.18,E2 11478.18} C_VEL
LIN {X 0,Y 574.791,Z 938.091,A -85,B 0,C 180,E1 11479.483,E2 11479.483} C_VEL
LIN {X 0,Y 541.058,Z 878.619,A -85,B 0,C 180,E1 11485.669,E2 11485.669} C_VEL
LIN {X 0,Y 514.238,Z 839.06,A -85,B 0,C 180,E1 11491.407,E2 11491.407} C_VEL
LIN {X 0,Y 513.96,Z 839.06,A -85,B 0,C 180,E1 11500.103,E2 11500.103} C_VEL
LIN {X 0,Y 514.391,Z 839.06,A -85,B 0,C 180,E1 11508.898,E2 11508.898} C_VEL
LIN {X 0,Y 515.44,Z 839.06,A -85,B 0,C 180,E1 11519.108,E2 11519.108} C_VEL
LIN {X 0,Y 514.497,Z 839.06,A -85,B 0,C 180,E1 11529.285,E2 11529.285} C_VEL
LIN {X 0,Y 514.028,Z 839.06,A -85,B 0,C 180,E1 11538.003,E2 11538.003} C_VEL
LIN {X 0,Y 513.926,Z 839.06,A -85,B 0,C 180,E1 11547.952,E2 11547.952} C_VEL
LIN {X 0,Y 514.201,Z 841.066,A -85,B 0,C 180,E1 11549.078,E2 11549.078} C_VEL
LIN {X 0,Y 549.089,Z 892.269,A -85,B 0,C 180,E1 11556.39,E2 11556.39} C_VEL
LIN {X 0,Y 573.566,Z 941.16,A -85,B 0,C 180,E1 11561.463,E2 11561.463} C_VEL
LIN {X 0,Y 562.35,Z 1014.859,A -85,B 0,C 180,E1 11564.692,E2 11564.692} C_VEL
LIN {X 0,Y 548.299,Z 1082.248,A -85,B 0,C 180,E1 11569.408,E2 11569.408} C_VEL
LIN {X 0,Y 534.178,Z 1142.209,A -85,B 0,C 180,E1 11575.747,E2 11575.747} C_VEL
LIN {X 0,Y 523.107,Z 1192.245,A -85,B 0,C 180,E1 11583.594,E2 11583.594} C_VEL
LIN {X 0,Y 517.389,Z 1227.895,A -85,B 0,C 180,E1 11592.055,E2 11592.055} C_VEL
LIN {X 0,Y 515.521,Z 1249.223,A -85,B 0,C 180,E1 11600.679,E2 11600.679} C_VEL
LIN {X 0,Y 515.064,Z 1256.407,A -85,B 0,C 180,E1 11607.466,E2 11607.466} C_VEL
LIN {X 0,Y 515.069,Z 1255.32,A -85,B 0,C 180,E1 11614.225,E2 11614.225} C_VEL
LIN {X 0,Y 515.488,Z 1244.058,A -85,B 0,C 180,E1 11621.896,E2 11621.896} C_VEL
LIN {X 0,Y 518.318,Z 1220.308,A -85,B 0,C 180,E1 11630.012,E2 11630.012} C_VEL
LIN {X 0,Y 525.712,Z 1180.355,A -85,B 0,C 180,E1 11638.455,E2 11638.455} C_VEL
LIN {X 0,Y 537.721,Z 1127.506,A -85,B 0,C 180,E1 11645.958,E2 11645.958} C_VEL
LIN {X 0,Y 552.068,Z 1065.19,A -85,B 0,C 180,E1 11651.896,E2 11651.896} C_VEL
LIN {X 0,Y 565.813,Z 995.514,A -85,B 0,C 180,E1 11656.225,E2 11656.225} C_VEL
LIN {X 0,Y 572.643,Z 938.882,A -85,B 0,C 180,E1 11658.652,E2 11658.652} C_VEL
LIN {X 0,Y 544.267,Z 884.125,A -85,B 0,C 180,E1 11664.472,E2 11664.472} C_VEL
LIN {X 0,Y 513.946,Z 839.06,A -85,B 0,C 180,E1 11671.193,E2 11671.193} C_VEL
LIN {X 0,Y 514.043,Z 839.06,A -85,B 0,C 180,E1 11680.21,E2 11680.21} C_VEL
LIN {X 0,Y 514.822,Z 839.06,A -85,B 0,C 180,E1 11689.006,E2 11689.006} C_VEL
LIN {X 0,Y 515.418,Z 839.06,A -85,B 0,C 180,E1 11699.205,E2 11699.205} C_VEL
LIN {X 0,Y 514.319,Z 839.06,A -85,B 0,C 180,E1 11709.386,E2 11709.386} C_VEL
LIN {X 0,Y 514.057,Z 839.06,A -85,B 0,C 180,E1 11718.104,E2 11718.104} C_VEL
LIN {X 0,Y 513.902,Z 839.06,A -85,B 0,C 180,E1 11727.951,E2 11727.951} C_VEL
LIN {X 0,Y 514.401,Z 841.755,A -85,B 0,C 180,E1 11728.744,E2 11728.744} C_VEL
LIN {X 0,Y 549.093,Z 891.333,A -85,B 0,C 180,E1 11735.828,E2 11735.828} C_VEL
LIN {X 0,Y 575.847,Z 942.064,A -85,B 0,C 180,E1 11740.784,E2 11740.784} C_VEL
LIN {X 0,Y 565.07,Z 1020.452,A -85,B 0,C 180,E1 11743.606,E2 11743.606} C_VEL
LIN {X 0,Y 551.596,Z 1091.676,A -85,B 0,C 180,E1 11747.972,E2 11747.972} C_VEL
LIN {X 0,Y 537.749,Z 1154.866,A -85,B 0,C 180,E1 11753.847,E2 11753.847} C_VEL
LIN {X 0,Y 526.171,Z 1207.95,A -85,B 0,C 180,E1 11761.101,E2 11761.101} C_VEL
LIN {X 0,Y 519.868,Z 1239.481,A -85,B 0,C 180,E1 11767.271,E2 11767.271} C_VEL
LIN {X 0,Y 510.288,Z 1254.09,A -85,B 0,C 180,E1 11770.725,E2 11770.725} C_VEL
LIN {X 0,Y 507.564,Z 1276.002,A -85,B 0,C 180,E1 11778.79,E2 11778.79} C_VEL
LIN {X 0,Y 506.993,Z 1285.348,A -85,B 0,C 180,E1 11785.707,E2 11785.707} C_VEL
LIN {X 0,Y 506.943,Z 1286.38,A -85,B 0,C 180,E1 11792.575,E2 11792.575} C_VEL
LIN {X 0,Y 507.645,Z 1277.568,A -85,B 0,C 180,E1 11800.337,E2 11800.337} C_VEL
LIN {X 0,Y 509.946,Z 1254.678,A -85,B 0,C 180,E1 11809.116,E2 11809.116} C_VEL
LIN {X 0,Y 516.36,Z 1218.635,A -85,B 0,C 180,E1 11817.442,E2 11817.442} C_VEL
LIN {X 0,Y 527.868,Z 1167.417,A -85,B 0,C 180,E1 11825.169,E2 11825.169} C_VEL
LIN {X 0,Y 542.305,Z 1105.324,A -85,B 0,C 180,E1 11831.505,E2 11831.505} C_VEL
LIN {X 0,Y 557.027,Z 1034.791,A -85,B 0,C 180,E1 11836.239,E2 11836.239} C_VEL
LIN {X 0,Y 568.595,Z 958.305,A -85,B 0,C 180,E1 11839.394,E2 11839.394} C_VEL
LIN {X 0,Y 569.186,Z 941.641,A -85,B 0,C 180,E1 11840.005,E2 11840.005} C_VEL
LIN {X 0,Y 537.103,Z 884.213,A -85,B 0,C 180,E1 11846.156,E2 11846.156} C_VEL
LIN {X 0,Y 506.164,Z 839.06,A -85,B 0,C 180,E1 11853.226,E2 11853.226} C_VEL
LIN {X 0,Y 506.174,Z 839.06,A -85,B 0,C 180,E1 11863.405,E2 11863.405} C_VEL
LIN {X 0,Y 506.634,Z 839.06,A -85,B 0,C 180,E1 11872.206,E2 11872.206} C_VEL
LIN {X 0,Y 506.819,Z 839.06,A -85,B 0,C 180,E1 11880.808,E2 11880.808} C_VEL
LIN {X 0,Y 506.459,Z 839.06,A -85,B 0,C 180,E1 11889.433,E2 11889.433} C_VEL
LIN {X 0,Y 505.961,Z 839.06,A -85,B 0,C 180,E1 11899.064,E2 11899.064} C_VEL
LIN {X 0,Y 506.19,Z 840.975,A -85,B 0,C 180,E1 11907.385,E2 11907.385} C_VEL
LIN {X 0,Y 541.028,Z 891.069,A -85,B 0,C 180,E1 11915.157,E2 11915.157} C_VEL
LIN {X 0,Y 567.897,Z 944.562,A -85,B 0,C 180,E1 11920.953,E2 11920.953} C_VEL
LIN {X 0,Y 555.819,Z 1019.619,A -85,B 0,C 180,E1 11924.344,E2 11924.344} C_VEL
LIN {X 0,Y 541.221,Z 1086.217,A -85,B 0,C 180,E1 11929.157,E2 11929.157} C_VEL
LIN {X 0,Y 526.718,Z 1145.011,A -85,B 0,C 180,E1 11935.561,E2 11935.561} C_VEL
LIN {X 0,Y 515.373,Z 1193.485,A -85,B 0,C 180,E1 11943.432,E2 11943.432} C_VEL
LIN {X 0,Y 509.493,Z 1227.893,A -85,B 0,C 180,E1 11951.768,E2 11951.768} C_VEL
LIN {X 0,Y 507.551,Z 1249.218,A -85,B 0,C 180,E1 11960.531,E2 11960.531} C_VEL
LIN {X 0,Y 507.085,Z 1256.407,A -85,B 0,C 180,E1 11967.426,E2 11967.426} C_VEL
LIN {X 0,Y 507.069,Z 1255.321,A -85,B 0,C 180,E1 11974.292,E2 11974.292} C_VEL
LIN {X 0,Y 507.566,Z 1244.059,A -85,B 0,C 180,E1 11982.085,E2 11982.085} C_VEL
LIN {X 0,Y 510.68,Z 1219.867,A -85,B 0,C 180,E1 11990.446,E2 11990.446} C_VEL
LIN {X 0,Y 518.781,Z 1179.172,A -85,B 0,C 180,E1 11999.11,E2 11999.11} C_VEL
LIN {X 0,Y 531.204,Z 1127.091,A -85,B 0,C 180,E1 12006.563,E2 12006.563} C_VEL
LIN {X 0,Y 545.986,Z 1065.292,A -85,B 0,C 180,E1 12012.489,E2 12012.489} C_VEL
LIN {X 0,Y 560.287,Z 995.354,A -85,B 0,C 180,E1 12016.847,E2 12016.847} C_VEL
LIN {X 0,Y 567,Z 942.289,A -85,B 0,C 180,E1 12019.164,E2 12019.164} C_VEL
LIN {X 0,Y 539.145,Z 888.241,A -85,B 0,C 180,E1 12025.133,E2 12025.133} C_VEL
LIN {X 0,Y 508.447,Z 844.851,A -85,B 0,C 180,E1 12031.893,E2 12031.893} C_VEL
LIN {X 0,Y 505.961,Z 839.06,A -85,B 0,C 180,E1 12032.843,E2 12032.843} C_VEL
LIN {X 0,Y 506.077,Z 839.06,A -85,B 0,C 180,E1 12041.704,E2 12041.704} C_VEL
LIN {X 0,Y 506.867,Z 839.06,A -85,B 0,C 180,E1 12050.574,E2 12050.574} C_VEL
LIN {X 0,Y 506.766,Z 839.06,A -85,B 0,C 180,E1 12060.907,E2 12060.907} C_VEL
LIN {X 0,Y 506.288,Z 839.06,A -85,B 0,C 180,E1 12069.537,E2 12069.537} C_VEL
LIN {X 0,Y 505.989,Z 839.06,A -85,B 0,C 180,E1 12079.076,E2 12079.076} C_VEL
LIN {X 0,Y 506.075,Z 840.618,A -85,B 0,C 180,E1 12086.96,E2 12086.96} C_VEL
LIN {X 0,Y 541.856,Z 891.848,A -85,B 0,C 180,E1 12094.78,E2 12094.78} C_VEL
LIN {X 0,Y 570.375,Z 944.203,A -85,B 0,C 180,E1 12100.232,E2 12100.232} C_VEL
LIN {X 0,Y 559.139,Z 1021.985,A -85,B 0,C 180,E1 12103.083,E2 12103.083} C_VEL
LIN {X 0,Y 544.957,Z 1093.615,A -85,B 0,C 180,E1 12107.553,E2 12107.553} C_VEL
LIN {X 0,Y 530.452,Z 1156.894,A -85,B 0,C 180,E1 12113.57,E2 12113.57} C_VEL
LIN {X 0,Y 518.322,Z 1210.516,A -85,B 0,C 180,E1 12121.101,E2 12121.101} C_VEL
LIN {X 0,Y 510.917,Z 1250.531,A -85,B 0,C 180,E1 12129.704,E2 12129.704} C_VEL
LIN {X 0,Y 510.288,Z 1254.09,A -85,B 0,C 180,E1 12130.725,E2 12130.725} C_VEL
LIN {X 0,Y 500.484,Z 1266.121,A -85,B 0,C 180,E1 12134.343,E2 12134.343} C_VEL
LIN {X 0,Y 499.44,Z 1282.873,A -85,B 0,C 180,E1 12143.017,E2 12143.017} C_VEL
LIN {X 0,Y 499.071,Z 1286.836,A -85,B 0,C 180,E1 12150.872,E2 12150.872} C_VEL
LIN {X 0,Y 499.244,Z 1280.557,A -85,B 0,C 180,E1 12158.683,E2 12158.683} C_VEL
LIN {X 0,Y 501.552,Z 1260.815,A -85,B 0,C 180,E1 12167.496,E2 12167.496} C_VEL
LIN {X 0,Y 507.615,Z 1226.096,A -85,B 0,C 180,E1 12176.372,E2 12176.372} C_VEL
LIN {X 0,Y 518.503,Z 1177.82,A -85,B 0,C 180,E1 12184.306,E2 12184.306} C_VEL
LIN {X 0,Y 533.136,Z 1117.804,A -85,B 0,C 180,E1 12190.979,E2 12190.979} C_VEL
LIN {X 0,Y 548.338,Z 1049.182,A -85,B 0,C 180,E1 12196.054,E2 12196.054} C_VEL
LIN {X 0,Y 561.556,Z 972.728,A -85,B 0,C 180,E1 12199.543,E2 12199.543} C_VEL
LIN {X 0,Y 563.598,Z 944.987,A -85,B 0,C 180,E1 12200.549,E2 12200.549} C_VEL
LIN {X 0,Y 532.198,Z 888.296,A -85,B 0,C 180,E1 12206.844,E2 12206.844} C_VEL
LIN {X 0,Y 501.578,Z 845.586,A -85,B 0,C 180,E1 12213.93,E2 12213.93} C_VEL
LIN {X 0,Y 498.042,Z 839.06,A -85,B 0,C 180,E1 12215.182,E2 12215.182} C_VEL
LIN {X 0,Y 498.159,Z 839.06,A -85,B 0,C 180,E1 12224.945,E2 12224.945} C_VEL
LIN {X 0,Y 498.449,Z 839.06,A -85,B 0,C 180,E1 12233.834,E2 12233.834} C_VEL
LIN {X 0,Y 498.811,Z 839.06,A -85,B 0,C 180,E1 12240.821,E2 12240.821} C_VEL
LIN {X 0,Y 498.436,Z 839.06,A -85,B 0,C 180,E1 12249.587,E2 12249.587} C_VEL
LIN {X 0,Y 497.966,Z 839.06,A -85,B 0,C 180,E1 12258.605,E2 12258.605} C_VEL
LIN {X 0,Y 498.141,Z 840.696,A -85,B 0,C 180,E1 12265.514,E2 12265.514} C_VEL
LIN {X 0,Y 531.012,Z 887.174,A -85,B 0,C 180,E1 12273.433,E2 12273.433} C_VEL
LIN {X 0,Y 559.537,Z 941.052,A -85,B 0,C 180,E1 12279.774,E2 12279.774} C_VEL
LIN {X 0,Y 561.603,Z 951.622,A -85,B 0,C 180,E1 12280.569,E2 12280.569} C_VEL
LIN {X 0,Y 548.733,Z 1026.091,A -85,B 0,C 180,E1 12284.105,E2 12284.105} C_VEL
LIN {X 0,Y 533.583,Z 1092.232,A -85,B 0,C 180,E1 12289.121,E2 12289.121} C_VEL
LIN {X 0,Y 518.698,Z 1149.616,A -85,B 0,C 180,E1 12295.65,E2 12295.65} C_VEL
LIN {X 0,Y 507.449,Z 1195.721,A -85,B 0,C 180,E1 12303.455,E2 12303.455} C_VEL
LIN {X 0,Y 501.45,Z 1230.098,A -85,B 0,C 180,E1 12312.212,E2 12312.212} C_VEL
LIN {X 0,Y 499.562,Z 1249.355,A -85,B 0,C 180,E1 12320.458,E2 12320.458} C_VEL
LIN {X 0,Y 499.085,Z 1256.407,A -85,B 0,C 180,E1 12327.384,E2 12327.384} C_VEL
LIN {X 0,Y 499.059,Z 1255.321,A -85,B 0,C 180,E1 12334.361,E2 12334.361} C_VEL
LIN {X 0,Y 499.646,Z 1244.06,A -85,B 0,C 180,E1 12342.279,E2 12342.279} C_VEL
LIN {X 0,Y 502.971,Z 1219.868,A -85,B 0,C 180,E1 12350.774,E2 12350.774} C_VEL
LIN {X 0,Y 511.912,Z 1178.141,A -85,B 0,C 180,E1 12359.784,E2 12359.784} C_VEL
LIN {X 0,Y 524.731,Z 1126.761,A -85,B 0,C 180,E1 12367.172,E2 12367.172} C_VEL
LIN {X 0,Y 540.231,Z 1064.169,A -85,B 0,C 180,E1 12373.191,E2 12373.191} C_VEL
LIN {X 0,Y 555.144,Z 993.66,A -85,B 0,C 180,E1 12377.55,E2 12377.55} C_VEL
LIN {X 0,Y 561.356,Z 945.799,A -85,B 0,C 180,E1 12379.682,E2 12379.682} C_VEL
LIN {X 0,Y 533.616,Z 891.26,A -85,B 0,C 180,E1 12385.894,E2 12385.894} C_VEL
LIN {X 0,Y 501.614,Z 845.781,A -85,B 0,C 180,E1 12393.378,E2 12393.378} C_VEL
LIN {X 0,Y 497.944,Z 839.06,A -85,B 0,C 180,E1 12394.806,E2 12394.806} C_VEL
LIN {X 0,Y 498.42,Z 839.06,A -85,B 0,C 180,E1 12405.057,E2 12405.057} C_VEL
LIN {X 0,Y 498.481,Z 839.06,A -85,B 0,C 180,E1 12413.935,E2 12413.935} C_VEL
LIN {X 0,Y 498.76,Z 839.06,A -85,B 0,C 180,E1 12420.922,E2 12420.922} C_VEL
LIN {X 0,Y 498.272,Z 839.06,A -85,B 0,C 180,E1 12429.692,E2 12429.692} C_VEL
LIN {X 0,Y 498.002,Z 839.06,A -85,B 0,C 180,E1 12438.709,E2 12438.709} C_VEL
LIN {X 0,Y 498.088,Z 840.671,A -85,B 0,C 180,E1 12445.117,E2 12445.117} C_VEL
LIN {X 0,Y 531.239,Z 887.063,A -85,B 0,C 180,E1 12452.98,E2 12452.98} C_VEL
LIN {X 0,Y 562.588,Z 942.712,A -85,B 0,C 180,E1 12459.244,E2 12459.244} C_VEL
LIN {X 0,Y 564.162,Z 953.626,A -85,B 0,C 180,E1 12459.88,E2 12459.88} C_VEL
LIN {X 0,Y 552.141,Z 1029.81,A -85,B 0,C 180,E1 12462.877,E2 12462.877} C_VEL
LIN {X 0,Y 537.285,Z 1099.903,A -85,B 0,C 180,E1 12467.472,E2 12467.472} C_VEL
LIN {X 0,Y 522.221,Z 1162.725,A -85,B 0,C 180,E1 12473.756,E2 12473.756} C_VEL
LIN {X 0,Y 510.039,Z 1214.663,A -85,B 0,C 180,E1 12481.447,E2 12481.447} C_VEL
LIN {X 0,Y 502.988,Z 1251.607,A -85,B 0,C 180,E1 12489.691,E2 12489.691} C_VEL
LIN {X 0,Y 500.484,Z 1266.121,A -85,B 0,C 180,E1 12494.343,E2 12494.343} C_VEL
LIN {X 0,Y 491.752,Z 1275.511,A -85,B 0,C 180,E1 12498.186,E2 12498.186} C_VEL
LIN {X 0,Y 491.002,Z 1285.347,A -85,B 0,C 180,E1 12505.567,E2 12505.567} C_VEL
LIN {X 0,Y 490.964,Z 1286.38,A -85,B 0,C 180,E1 12512.659,E2 12512.659} C_VEL
LIN {X 0,Y 491.71,Z 1277.563,A -85,B 0,C 180,E1 12520.676,E2 12520.676} C_VEL
LIN {X 0,Y 494.248,Z 1254.902,A -85,B 0,C 180,E1 12529.679,E2 12529.679} C_VEL
LIN {X 0,Y 501.059,Z 1219.853,A -85,B 0,C 180,E1 12538.01,E2 12538.01} C_VEL
LIN {X 0,Y 513.625,Z 1169.049,A -85,B 0,C 180,E1 12545.975,E2 12545.975} C_VEL
LIN {X 0,Y 529.392,Z 1107.064,A -85,B 0,C 180,E1 12552.505,E2 12552.505} C_VEL
LIN {X 0,Y 545.107,Z 1037.678,A -85,B 0,C 180,E1 12557.302,E2 12557.302} C_VEL
LIN {X 0,Y 557.809,Z 960.657,A -85,B 0,C 180,E1 12560.57,E2 12560.57} C_VEL
LIN {X 0,Y 557.824,Z 947.893,A -85,B 0,C 180,E1 12561.151,E2 12561.151} C_VEL
LIN {X 0,Y 527.105,Z 891.881,A -85,B 0,C 180,E1 12567.587,E2 12567.587} C_VEL
LIN {X 0,Y 498.137,Z 851.786,A -85,B 0,C 180,E1 12574.54,E2 12574.54} C_VEL
LIN {X 0,Y 489.921,Z 839.06,A -85,B 0,C 180,E1 12577.171,E2 12577.171} C_VEL
LIN {X 0,Y 490.214,Z 839.06,A -85,B 0,C 180,E1 12587.295,E2 12587.295} C_VEL
LIN {X 0,Y 490.808,Z 839.06,A -85,B 0,C 180,E1 12597.291,E2 12597.291} C_VEL
LIN {X 0,Y 490.657,Z 839.06,A -85,B 0,C 180,E1 12607.947,E2 12607.947} C_VEL
LIN {X 0,Y 490.053,Z 839.06,A -85,B 0,C 180,E1 12617.051,E2 12617.051} C_VEL
LIN {X 0,Y 490.157,Z 841.057,A -85,B 0,C 180,E1 12623.475,E2 12623.475} C_VEL
LIN {X 0,Y 519.423,Z 881.067,A -85,B 0,C 180,E1 12631.234,E2 12631.234} C_VEL
LIN {X 0,Y 547.946,Z 931.408,A -85,B 0,C 180,E1 12637.79,E2 12637.79} C_VEL
LIN {X 0,Y 556.04,Z 954.206,A -85,B 0,C 180,E1 12640.021,E2 12640.021} C_VEL
LIN {X 0,Y 542.487,Z 1029.096,A -85,B 0,C 180,E1 12643.656,E2 12643.656} C_VEL
LIN {X 0,Y 526.467,Z 1095.921,A -85,B 0,C 180,E1 12648.86,E2 12648.86} C_VEL
LIN {X 0,Y 510.93,Z 1153.398,A -85,B 0,C 180,E1 12655.629,E2 12655.629} C_VEL
LIN {X 0,Y 499.188,Z 1199.726,A -85,B 0,C 180,E1 12663.834,E2 12663.834} C_VEL
LIN {X 0,Y 493.302,Z 1233.261,A -85,B 0,C 180,E1 12673,E2 12673} C_VEL
LIN {X 0,Y 491.256,Z 1251.742,A -85,B 0,C 180,E1 12682.006,E2 12682.006} C_VEL
LIN {X 0,Y 490.795,Z 1256.845,A -85,B 0,C 180,E1 12689.113,E2 12689.113} C_VEL
LIN {X 0,Y 491.261,Z 1252.819,A -85,B 0,C 180,E1 12697.1,E2 12697.1} C_VEL
LIN {X 0,Y 492.914,Z 1235.534,A -85,B 0,C 180,E1 12706.092,E2 12706.092} C_VEL
LIN {X 0,Y 498.281,Z 1203.517,A -85,B 0,C 180,E1 12715.248,E2 12715.248} C_VEL
LIN {X 0,Y 509.402,Z 1159.104,A -85,B 0,C 180,E1 12723.458,E2 12723.458} C_VEL
LIN {X 0,Y 524.792,Z 1102.104,A -85,B 0,C 180,E1 12730.466,E2 12730.466} C_VEL
LIN {X 0,Y 541.088,Z 1036.144,A -85,B 0,C 180,E1 12735.802,E2 12735.802} C_VEL
LIN {X 0,Y 554.888,Z 962.666,A -85,B 0,C 180,E1 12739.565,E2 12739.565} C_VEL
LIN {X 0,Y 555.429,Z 948.515,A -85,B 0,C 180,E1 12740.275,E2 12740.275} C_VEL
LIN {X 0,Y 528.723,Z 895.741,A -85,B 0,C 180,E1 12746.526,E2 12746.526} C_VEL
LIN {X 0,Y 498.795,Z 852.607,A -85,B 0,C 180,E1 12753.818,E2 12753.818} C_VEL
LIN {X 0,Y 489.915,Z 839.06,A -85,B 0,C 180,E1 12756.721,E2 12756.721} C_VEL
LIN {X 0,Y 490.586,Z 839.06,A -85,B 0,C 180,E1 12767.099,E2 12767.099} C_VEL
LIN {X 0,Y 490.425,Z 839.06,A -85,B 0,C 180,E1 12775.615,E2 12775.615} C_VEL
LIN {X 0,Y 490.538,Z 839.06,A -85,B 0,C 180,E1 12782.71,E2 12782.71} C_VEL
LIN {X 0,Y 490.159,Z 839.06,A -85,B 0,C 180,E1 12791.659,E2 12791.659} C_VEL
LIN {X 0,Y 489.958,Z 839.06,A -85,B 0,C 180,E1 12800.916,E2 12800.916} C_VEL
LIN {X 0,Y 490.106,Z 840.669,A -85,B 0,C 180,E1 12803.071,E2 12803.071} C_VEL
LIN {X 0,Y 519.932,Z 881.645,A -85,B 0,C 180,E1 12810.885,E2 12810.885} C_VEL
LIN {X 0,Y 550.325,Z 932.548,A -85,B 0,C 180,E1 12817.269,E2 12817.269} C_VEL
LIN {X 0,Y 558.876,Z 954.293,A -85,B 0,C 180,E1 12819.271,E2 12819.271} C_VEL
LIN {X 0,Y 546.356,Z 1030.562,A -85,B 0,C 180,E1 12822.298,E2 12822.298} C_VEL
LIN {X 0,Y 530.827,Z 1100.938,A -85,B 0,C 180,E1 12826.973,E2 12826.973} C_VEL
LIN {X 0,Y 515.107,Z 1163.679,A -85,B 0,C 180,E1 12833.356,E2 12833.356} C_VEL
LIN {X 0,Y 502.468,Z 1215.078,A -85,B 0,C 180,E1 12841.115,E2 12841.115} C_VEL
LIN {X 0,Y 494.945,Z 1253.142,A -85,B 0,C 180,E1 12849.815,E2 12849.815} C_VEL
LIN {X 0,Y 491.752,Z 1275.511,A -85,B 0,C 180,E1 12858.186,E2 12858.186} C_VEL
LIN {X 0,Y 483.372,Z 1282.062,A -85,B 0,C 180,E1 12862.168,E2 12862.168} C_VEL
LIN {X 0,Y 483.076,Z 1286.836,A -85,B 0,C 180,E1 12870.901,E2 12870.901} C_VEL
LIN {X 0,Y 483.321,Z 1280.465,A -85,B 0,C 180,E1 12879.036,E2 12879.036} C_VEL
LIN {X 0,Y 485.874,Z 1260.391,A -85,B 0,C 180,E1 12888.228,E2 12888.228} C_VEL
LIN {X 0,Y 492.502,Z 1225.338,A -85,B 0,C 180,E1 12897.292,E2 12897.292} C_VEL
LIN {X 0,Y 504.522,Z 1177.387,A -85,B 0,C 180,E1 12905.377,E2 12905.377} C_VEL
LIN {X 0,Y 520.45,Z 1117.784,A -85,B 0,C 180,E1 12912.14,E2 12912.14} C_VEL
LIN {X 0,Y 536.823,Z 1049.67,A -85,B 0,C 180,E1 12917.256,E2 12917.256} C_VEL
LIN {X 0,Y 550.923,Z 973.511,A -85,B 0,C 180,E1 12920.786,E2 12920.786} C_VEL
LIN {X 0,Y 552.39,Z 951.753,A -85,B 0,C 180,E1 12921.668,E2 12921.668} C_VEL
LIN {X 0,Y 523.121,Z 897.39,A -85,B 0,C 180,E1 12928.108,E2 12928.108} C_VEL
LIN {X 0,Y 495.406,Z 858.456,A -85,B 0,C 180,E1 12934.983,E2 12934.983} C_VEL
LIN {X 0,Y 481.882,Z 839.06,A -85,B 0,C 180,E1 12939.682,E2 12939.682} C_VEL
LIN {X 0,Y 482.505,Z 839.06,A -85,B 0,C 180,E1 12949.989,E2 12949.989} C_VEL
LIN {X 0,Y 482.82,Z 839.06,A -85,B 0,C 180,E1 12960.849,E2 12960.849} C_VEL
LIN {X 0,Y 482.379,Z 839.06,A -85,B 0,C 180,E1 12969.909,E2 12969.909} C_VEL
LIN {X 0,Y 481.904,Z 839.06,A -85,B 0,C 180,E1 12980.207,E2 12980.207} C_VEL
LIN {X 0,Y 482.382,Z 841.692,A -85,B 0,C 180,E1 12981.25,E2 12981.25} C_VEL
LIN {X 0,Y 505.035,Z 871.519,A -85,B 0,C 180,E1 12988.061,E2 12988.061} C_VEL
LIN {X 0,Y 533.266,Z 916.493,A -85,B 0,C 180,E1 12994.956,E2 12994.956} C_VEL
LIN {X 0,Y 550.694,Z 955.78,A -85,B 0,C 180,E1 12999.428,E2 12999.428} C_VEL
LIN {X 0,Y 536.506,Z 1031.059,A -85,B 0,C 180,E1 13003.132,E2 13003.132} C_VEL
LIN {X 0,Y 520.098,Z 1096.845,A -85,B 0,C 180,E1 13008.326,E2 13008.326} C_VEL
LIN {X 0,Y 504.038,Z 1153.668,A -85,B 0,C 180,E1 13015.091,E2 13015.091} C_VEL
LIN {X 0,Y 491.712,Z 1199.996,A -85,B 0,C 180,E1 13023.405,E2 13023.405} C_VEL
LIN {X 0,Y 485.412,Z 1233.258,A -85,B 0,C 180,E1 13032.715,E2 13032.715} C_VEL
LIN {X 0,Y 483.282,Z 1251.738,A -85,B 0,C 180,E1 13041.873,E2 13041.873} C_VEL
LIN {X 0,Y 482.796,Z 1256.844,A -85,B 0,C 180,E1 13049.099,E2 13049.099} C_VEL
LIN {X 0,Y 483.289,Z 1252.82,A -85,B 0,C 180,E1 13057.218,E2 13057.218} C_VEL
LIN {X 0,Y 484.986,Z 1235.536,A -85,B 0,C 180,E1 13066.362,E2 13066.362} C_VEL
LIN {X 0,Y 490.358,Z 1205.702,A -85,B 0,C 180,E1 13075.194,E2 13075.194} C_VEL
LIN {X 0,Y 501.577,Z 1162.453,A -85,B 0,C 180,E1 13083.494,E2 13083.494} C_VEL
LIN {X 0,Y 517.28,Z 1106.882,A -85,B 0,C 180,E1 13090.585,E2 13090.585} C_VEL
LIN {X 0,Y 533.868,Z 1042.765,A -85,B 0,C 180,E1 13096.004,E2 13096.004} C_VEL
LIN {X 0,Y 548.331,Z 970.419,A -85,B 0,C 180,E1 13099.915,E2 13099.915} C_VEL
LIN {X 0,Y 549.815,Z 952.205,A -85,B 0,C 180,E1 13100.792,E2 13100.792} C_VEL
LIN {X 0,Y 523.924,Z 900.046,A -85,B 0,C 180,E1 13107.171,E2 13107.171} C_VEL
LIN {X 0,Y 495.713,Z 859.05,A -85,B 0,C 180,E1 13114.347,E2 13114.347} C_VEL
LIN {X 0,Y 481.999,Z 839.06,A -85,B 0,C 180,E1 13119.316,E2 13119.316} C_VEL
LIN {X 0,Y 482.7,Z 839.06,A -85,B 0,C 180,E1 13128.264,E2 13128.264} C_VEL
LIN {X 0,Y 483.363,Z 839.06,A -85,B 0,C 180,E1 13139.152,E2 13139.152} C_VEL
LIN {X 0,Y 482.225,Z 839.06,A -85,B 0,C 180,E1 13150.017,E2 13150.017} C_VEL
LIN {X 0,Y 481.947,Z 839.06,A -85,B 0,C 180,E1 13159.357,E2 13159.357} C_VEL
LIN {X 0,Y 482.289,Z 841.365,A -85,B 0,C 180,E1 13160.842,E2 13160.842} C_VEL
LIN {X 0,Y 507.689,Z 874.711,A -85,B 0,C 180,E1 13168.316,E2 13168.316} C_VEL
LIN {X 0,Y 539.187,Z 924.921,A -85,B 0,C 180,E1 13175.408,E2 13175.408} C_VEL
LIN {X 0,Y 553.341,Z 957.418,A -85,B 0,C 180,E1 13178.726,E2 13178.726} C_VEL
LIN {X 0,Y 540.124,Z 1033.971,A -85,B 0,C 180,E1 13181.856,E2 13181.856} C_VEL
LIN {X 0,Y 523.797,Z 1104.345,A -85,B 0,C 180,E1 13186.662,E2 13186.662} C_VEL
LIN {X 0,Y 507.395,Z 1166.995,A -85,B 0,C 180,E1 13193.246,E2 13193.246} C_VEL
LIN {X 0,Y 494.478,Z 1217.651,A -85,B 0,C 180,E1 13201.187,E2 13201.187} C_VEL
LIN {X 0,Y 486.89,Z 1254.751,A -85,B 0,C 180,E1 13209.965,E2 13209.965} C_VEL
LIN {X 0,Y 483.499,Z 1277.561,A -85,B 0,C 180,E1 13219.142,E2 13219.142} C_VEL
LIN {X 0,Y 483.372,Z 1282.062,A -85,B 0,C 180,E1 13222.168,E2 13222.168} C_VEL
LIN {X 0,Y 475.003,Z 1285.823,A -85,B 0,C 180,E1 13226.264,E2 13226.264} C_VEL
LIN {X 0,Y 475.19,Z 1285.347,A -85,B 0,C 180,E1 13234.582,E2 13234.582} C_VEL
LIN {X 0,Y 475.927,Z 1273.354,A -85,B 0,C 180,E1 13243.292,E2 13243.292} C_VEL
LIN {X 0,Y 479.121,Z 1251.259,A -85,B 0,C 180,E1 13251.37,E2 13251.37} C_VEL
LIN {X 0,Y 487.483,Z 1214.387,A -85,B 0,C 180,E1 13259.886,E2 13259.886} C_VEL
LIN {X 0,Y 501.473,Z 1163.332,A -85,B 0,C 180,E1 13267.779,E2 13267.779} C_VEL
LIN {X 0,Y 518.64,Z 1101.248,A -85,B 0,C 180,E1 13274.202,E2 13274.202} C_VEL
LIN {X 0,Y 534.882,Z 1033.734,A -85,B 0,C 180,E1 13278.776,E2 13278.776} C_VEL
LIN {X 0,Y 547.173,Z 956.123,A -85,B 0,C 180,E1 13282.139,E2 13282.139} C_VEL
LIN {X 0,Y 519.612,Z 903.441,A -85,B 0,C 180,E1 13288.544,E2 13288.544} C_VEL
LIN {X 0,Y 490.343,Z 861.186,A -85,B 0,C 180,E1 13296.173,E2 13296.173} C_VEL
LIN {X 0,Y 473.982,Z 839.06,A -85,B 0,C 180,E1 13302.241,E2 13302.241} C_VEL
LIN {X 0,Y 474.585,Z 839.06,A -85,B 0,C 180,E1 13311.676,E2 13311.676} C_VEL
LIN {X 0,Y 474.812,Z 839.06,A -85,B 0,C 180,E1 13320.863,E2 13320.863} C_VEL
LIN {X 0,Y 474.346,Z 839.06,A -85,B 0,C 180,E1 13330.079,E2 13330.079} C_VEL
LIN {X 0,Y 474.116,Z 840.83,A -85,B 0,C 180,E1 13338.437,E2 13338.437} C_VEL
LIN {X 0,Y 496.8,Z 870.529,A -85,B 0,C 180,E1 13346.167,E2 13346.167} C_VEL
LIN {X 0,Y 524.818,Z 914.262,A -85,B 0,C 180,E1 13353.485,E2 13353.485} C_VEL
LIN {X 0,Y 545.136,Z 959.135,A -85,B 0,C 180,E1 13358.889,E2 13358.889} C_VEL
LIN {X 0,Y 530.444,Z 1033.591,A -85,B 0,C 180,E1 13362.631,E2 13362.631} C_VEL
LIN {X 0,Y 513.376,Z 1099.195,A -85,B 0,C 180,E1 13367.916,E2 13367.916} C_VEL
LIN {X 0,Y 496.782,Z 1155.514,A -85,B 0,C 180,E1 13374.773,E2 13374.773} C_VEL
LIN {X 0,Y 484.078,Z 1201.185,A -85,B 0,C 180,E1 13383.169,E2 13383.169} C_VEL
LIN {X 0,Y 477.509,Z 1233.326,A -85,B 0,C 180,E1 13392.42,E2 13392.42} C_VEL
LIN {X 0,Y 475.321,Z 1251.734,A -85,B 0,C 180,E1 13401.736,E2 13401.736} C_VEL
LIN {X 0,Y 474.814,Z 1256.844,A -85,B 0,C 180,E1 13409.083,E2 13409.083} C_VEL
LIN {X 0,Y 475.299,Z 1252.821,A -85,B 0,C 180,E1 13417.34,E2 13417.34} C_VEL
LIN {X 0,Y 477.053,Z 1235.554,A -85,B 0,C 180,E1 13426.642,E2 13426.642} C_VEL
LIN {X 0,Y 482.776,Z 1206.2,A -85,B 0,C 180,E1 13435.56,E2 13435.56} C_VEL
LIN {X 0,Y 494.415,Z 1163.553,A -85,B 0,C 180,E1 13443.893,E2 13443.893} C_VEL
LIN {X 0,Y 510.897,Z 1107.644,A -85,B 0,C 180,E1 13451.135,E2 13451.135} C_VEL
LIN {X 0,Y 528.204,Z 1043.165,A -85,B 0,C 180,E1 13456.632,E2 13456.632} C_VEL
LIN {X 0,Y 543.238,Z 970.502,A -85,B 0,C 180,E1 13460.57,E2 13460.57} C_VEL
LIN {X 0,Y 544.547,Z 956.621,A -85,B 0,C 180,E1 13461.238,E2 13461.238} C_VEL
LIN {X 0,Y 519.193,Z 904.348,A -85,B 0,C 180,E1 13467.828,E2 13467.828} C_VEL
LIN {X 0,Y 489.839,Z 860.844,A -85,B 0,C 180,E1 13475.771,E2 13475.771} C_VEL
LIN {X 0,Y 473.995,Z 839.06,A -85,B 0,C 180,E1 13481.668,E2 13481.668} C_VEL
LIN {X 0,Y 474.713,Z 839.06,A -85,B 0,C 180,E1 13491.784,E2 13491.784} C_VEL
LIN {X 0,Y 474.769,Z 839.06,A -85,B 0,C 180,E1 13500.968,E2 13500.968} C_VEL
LIN {X 0,Y 474.198,Z 839.06,A -85,B 0,C 180,E1 13510.189,E2 13510.189} C_VEL
LIN {X 0,Y 474.153,Z 840.804,A -85,B 0,C 180,E1 13518.099,E2 13518.099} C_VEL
LIN {X 0,Y 497.041,Z 870.954,A -85,B 0,C 180,E1 13525.853,E2 13525.853} C_VEL
LIN {X 0,Y 527.091,Z 916.131,A -85,B 0,C 180,E1 13533.211,E2 13533.211} C_VEL
LIN {X 0,Y 547.919,Z 960.136,A -85,B 0,C 180,E1 13538.159,E2 13538.159} C_VEL
LIN {X 0,Y 534.353,Z 1035.139,A -85,B 0,C 180,E1 13541.277,E2 13541.277} C_VEL
LIN {X 0,Y 517.176,Z 1106.273,A -85,B 0,C 180,E1 13546.217,E2 13546.217} C_VEL
LIN {X 0,Y 500.672,Z 1166.718,A -85,B 0,C 180,E1 13552.669,E2 13552.669} C_VEL
LIN {X 0,Y 486.917,Z 1218.023,A -85,B 0,C 180,E1 13560.831,E2 13560.831} C_VEL
LIN {X 0,Y 478.96,Z 1255.278,A -85,B 0,C 180,E1 13569.856,E2 13569.856} C_VEL
LIN {X 0,Y 475.556,Z 1277.558,A -85,B 0,C 180,E1 13578.958,E2 13578.958} C_VEL
LIN {X 0,Y 475.003,Z 1285.823,A -85,B 0,C 180,E1 13586.264,E2 13586.264} C_VEL
LIN {X 0,Y 467.133,Z 1286.836,A -85,B 0,C 180,E1 13590.5,E2 13590.5} C_VEL
LIN {X 0,Y 467.397,Z 1280.459,A -85,B 0,C 180,E1 13599.347,E2 13599.347} C_VEL
LIN {X 0,Y 470.128,Z 1260.067,A -85,B 0,C 180,E1 13608.84,E2 13608.84} C_VEL
LIN {X 0,Y 477.406,Z 1225.089,A -85,B 0,C 180,E1 13618.159,E2 13618.159} C_VEL
LIN {X 0,Y 490.761,Z 1177.07,A -85,B 0,C 180,E1 13626.486,E2 13626.486} C_VEL
LIN {X 0,Y 508.127,Z 1117.276,A -85,B 0,C 180,E1 13633.406,E2 13633.406} C_VEL
LIN {X 0,Y 525.737,Z 1049.248,A -85,B 0,C 180,E1 13638.57,E2 13638.57} C_VEL
LIN {X 0,Y 540.593,Z 974.088,A -85,B 0,C 180,E1 13642.084,E2 13642.084} C_VEL
LIN {X 0,Y 541.419,Z 959.042,A -85,B 0,C 180,E1 13642.768,E2 13642.768} C_VEL
LIN {X 0,Y 513.912,Z 905.779,A -85,B 0,C 180,E1 13649.513,E2 13649.513} C_VEL
LIN {X 0,Y 487.011,Z 867.551,A -85,B 0,C 180,E1 13656.834,E2 13656.834} C_VEL
LIN {X 0,Y 469.505,Z 845.669,A -85,B 0,C 180,E1 13663.52,E2 13663.52} C_VEL
LIN {X 0,Y 466.092,Z 839.06,A -85,B 0,C 180,E1 13665.814,E2 13665.814} C_VEL
LIN {X 0,Y 466.452,Z 839.06,A -85,B 0,C 180,E1 13675.282,E2 13675.282} C_VEL
LIN {X 0,Y 466.515,Z 839.06,A -85,B 0,C 180,E1 13682.743,E2 13682.743} C_VEL
LIN {X 0,Y 466.241,Z 839.06,A -85,B 0,C 180,E1 13692.156,E2 13692.156} C_VEL
LIN {X 0,Y 466.426,Z 841.214,A -85,B 0,C 180,E1 13695.33,E2 13695.33} C_VEL
LIN {X 0,Y 484.328,Z 864.287,A -85,B 0,C 180,E1 13702.713,E2 13702.713} C_VEL
LIN {X 0,Y 509.943,Z 901.149,A -85,B 0,C 180,E1 13710.203,E2 13710.203} C_VEL
LIN {X 0,Y 534.474,Z 948.81,A -85,B 0,C 180,E1 13716.788,E2 13716.788} C_VEL
LIN {X 0,Y 539.251,Z 964.908,A -85,B 0,C 180,E1 13718.429,E2 13718.429} C_VEL
LIN {X 0,Y 523.593,Z 1039.338,A -85,B 0,C 180,E1 13722.323,E2 13722.323} C_VEL
LIN {X 0,Y 505.595,Z 1105.245,A -85,B 0,C 180,E1 13727.874,E2 13727.874} C_VEL
LIN {X 0,Y 488.334,Z 1161.558,A -85,B 0,C 180,E1 13735.109,E2 13735.109} C_VEL
LIN {X 0,Y 475.692,Z 1205.4,A -85,B 0,C 180,E1 13743.657,E2 13743.657} C_VEL
LIN {X 0,Y 469.399,Z 1236.112,A -85,B 0,C 180,E1 13753.115,E2 13753.115} C_VEL
LIN {X 0,Y 467.221,Z 1252.92,A -85,B 0,C 180,E1 13762.532,E2 13762.532} C_VEL
LIN {X 0,Y 467.136,Z 1256.827,A -85,B 0,C 180,E1 13770.93,E2 13770.93} C_VEL
LIN {X 0,Y 467.468,Z 1250.523,A -85,B 0,C 180,E1 13779.25,E2 13779.25} C_VEL
LIN {X 0,Y 469.574,Z 1232.057,A -85,B 0,C 180,E1 13788.373,E2 13788.373} C_VEL
LIN {X 0,Y 476.452,Z 1201.853,A -85,B 0,C 180,E1 13797.112,E2 13797.112} C_VEL
LIN {X 0,Y 489.606,Z 1156.956,A -85,B 0,C 180,E1 13805.528,E2 13805.528} C_VEL
LIN {X 0,Y 507.235,Z 1099.226,A -85,B 0,C 180,E1 13812.651,E2 13812.651} C_VEL
LIN {X 0,Y 524.875,Z 1034.562,A -85,B 0,C 180,E1 13817.873,E2 13817.873} C_VEL
LIN {X 0,Y 538.883,Z 959.758,A -85,B 0,C 180,E1 13821.828,E2 13821.828} C_VEL
LIN {X 0,Y 514.347,Z 908.588,A -85,B 0,C 180,E1 13828.533,E2 13828.533} C_VEL
LIN {X 0,Y 487.346,Z 867.901,A -85,B 0,C 180,E1 13836.183,E2 13836.183} C_VEL
LIN {X 0,Y 469.592,Z 845.648,A -85,B 0,C 180,E1 13842.902,E2 13842.902} C_VEL
LIN {X 0,Y 466.294,Z 839.06,A -85,B 0,C 180,E1 13844.968,E2 13844.968} C_VEL
LIN {X 0,Y 466.512,Z 839.06,A -85,B 0,C 180,E1 13853.518,E2 13853.518} C_VEL
LIN {X 0,Y 466.762,Z 839.06,A -85,B 0,C 180,E1 13860.985,E2 13860.985} C_VEL
LIN {X 0,Y 466.176,Z 839.06,A -85,B 0,C 180,E1 13870.366,E2 13870.366} C_VEL
LIN {X 0,Y 466.347,Z 841.085,A -85,B 0,C 180,E1 13874.96,E2 13874.96} C_VEL
LIN {X 0,Y 484.121,Z 863.99,A -85,B 0,C 180,E1 13882.271,E2 13882.271} C_VEL
LIN {X 0,Y 510.978,Z 901.76,A -85,B 0,C 180,E1 13889.819,E2 13889.819} C_VEL
LIN {X 0,Y 537.973,Z 951.404,A -85,B 0,C 180,E1 13896.375,E2 13896.375} C_VEL
LIN {X 0,Y 542.236,Z 965.438,A -85,B 0,C 180,E1 13897.666,E2 13897.666} C_VEL
LIN {X 0,Y 527.784,Z 1040.568,A -85,B 0,C 180,E1 13900.926,E2 13900.926} C_VEL
LIN {X 0,Y 510.092,Z 1110.042,A -85,B 0,C 180,E1 13905.92,E2 13905.92} C_VEL
LIN {X 0,Y 492.806,Z 1170.58,A -85,B 0,C 180,E1 13912.615,E2 13912.615} C_VEL
LIN {X 0,Y 479.051,Z 1219.981,A -85,B 0,C 180,E1 13920.779,E2 13920.779} C_VEL
LIN {X 0,Y 470.729,Z 1257.302,A -85,B 0,C 180,E1 13930.207,E2 13930.207} C_VEL
LIN {X 0,Y 467.601,Z 1277.555,A -85,B 0,C 180,E1 13938.768,E2 13938.768} C_VEL
LIN {X 0,Y 467.079,Z 1286.38,A -85,B 0,C 180,E1 13947.206,E2 13947.206} C_VEL
LIN {X 0,Y 467.133,Z 1286.836,A -85,B 0,C 180,E1 13950.5,E2 13950.5} C_VEL
LIN {X 0,Y 459.184,Z 1285.317,A -85,B 0,C 180,E1 13954.777,E2 13954.777} C_VEL
LIN {X 0,Y 459.975,Z 1273.455,A -85,B 0,C 180,E1 13963.556,E2 13963.556} C_VEL
LIN {X 0,Y 463.595,Z 1250.711,A -85,B 0,C 180,E1 13972.123,E2 13972.123} C_VEL
LIN {X 0,Y 472.88,Z 1213.831,A -85,B 0,C 180,E1 13980.908,E2 13980.908} C_VEL
LIN {X 0,Y 488.562,Z 1161.586,A -85,B 0,C 180,E1 13989.154,E2 13989.154} C_VEL
LIN {X 0,Y 507.137,Z 1099.552,A -85,B 0,C 180,E1 13995.618,E2 13995.618} C_VEL
LIN {X 0,Y 524.586,Z 1031.624,A -85,B 0,C 180,E1 14000.21,E2 14000.21} C_VEL
LIN {X 0,Y 536.019,Z 962.836,A -85,B 0,C 180,E1 14003.326,E2 14003.326} C_VEL
LIN {X 0,Y 510.069,Z 911.63,A -85,B 0,C 180,E1 14009.999,E2 14009.999} C_VEL
LIN {X 0,Y 484.921,Z 874.867,A -85,B 0,C 180,E1 14017.14,E2 14017.14} C_VEL
LIN {X 0,Y 467.047,Z 852.489,A -85,B 0,C 180,E1 14024.181,E2 14024.181} C_VEL
LIN {X 0,Y 461.312,Z 845.411,A -85,B 0,C 180,E1 14027.36,E2 14027.36} C_VEL
LIN {X 0,Y 458.442,Z 839.06,A -85,B 0,C 180,E1 14030.42,E2 14030.42} C_VEL
LIN {X 0,Y 458.796,Z 839.06,A -85,B 0,C 180,E1 14040.893,E2 14040.893} C_VEL
LIN {X 0,Y 458.307,Z 840.091,A -85,B 0,C 180,E1 14050.857,E2 14050.857} C_VEL
LIN {X 0,Y 470.927,Z 856.92,A -85,B 0,C 180,E1 14058.023,E2 14058.023} C_VEL
LIN {X 0,Y 492.03,Z 885.054,A -85,B 0,C 180,E1 14065.58,E2 14065.58} C_VEL
LIN {X 0,Y 518.182,Z 928.6,A -85,B 0,C 180,E1 14073.056,E2 14073.056} C_VEL
LIN {X 0,Y 533.812,Z 967.586,A -85,B 0,C 180,E1 14077.849,E2 14077.849} C_VEL
LIN {X 0,Y 517.702,Z 1041.146,A -85,B 0,C 180,E1 14081.762,E2 14081.762} C_VEL
LIN {X 0,Y 499.052,Z 1106.838,A -85,B 0,C 180,E1 14087.38,E2 14087.38} C_VEL
LIN {X 0,Y 481.196,Z 1162.771,A -85,B 0,C 180,E1 14094.696,E2 14094.696} C_VEL
LIN {X 0,Y 468.034,Z 1206.393,A -85,B 0,C 180,E1 14103.389,E2 14103.389} C_VEL
LIN {X 0,Y 461.511,Z 1236.555,A -85,B 0,C 180,E1 14112.895,E2 14112.895} C_VEL
LIN {X 0,Y 459.236,Z 1253.1,A -85,B 0,C 180,E1 14122.523,E2 14122.523} C_VEL
LIN {X 0,Y 459.164,Z 1256.827,A -85,B 0,C 180,E1 14130.947,E2 14130.947} C_VEL
LIN {X 0,Y 459.481,Z 1249.237,A -85,B 0,C 180,E1 14140.469,E2 14140.469} C_VEL
LIN {X 0,Y 461.997,Z 1231.024,A -85,B 0,C 180,E1 14149.183,E2 14149.183} C_VEL
LIN {X 0,Y 470.258,Z 1198.317,A -85,B 0,C 180,E1 14158.435,E2 14158.435} C_VEL
LIN {X 0,Y 484.848,Z 1150.958,A -85,B 0,C 180,E1 14167.04,E2 14167.04} C_VEL
LIN {X 0,Y 503.43,Z 1092.041,A -85,B 0,C 180,E1 14174.026,E2 14174.026} C_VEL
LIN {X 0,Y 521.792,Z 1025.299,A -85,B 0,C 180,E1 14179.138,E2 14179.138} C_VEL
LIN {X 0,Y 533.446,Z 963.609,A -85,B 0,C 180,E1 14182.362,E2 14182.362} C_VEL
LIN {X 0,Y 509.24,Z 912.13,A -85,B 0,C 180,E1 14189.318,E2 14189.318} C_VEL
LIN {X 0,Y 484.002,Z 873.957,A -85,B 0,C 180,E1 14196.865,E2 14196.865} C_VEL
LIN {X 0,Y 466.934,Z 852.318,A -85,B 0,C 180,E1 14203.648,E2 14203.648} C_VEL
LIN {X 0,Y 461.92,Z 845.634,A -85,B 0,C 180,E1 14206.401,E2 14206.401} C_VEL
LIN {X 0,Y 458.709,Z 839.06,A -85,B 0,C 180,E1 14209.574,E2 14209.574} C_VEL
LIN {X 0,Y 459.314,Z 839.06,A -85,B 0,C 180,E1 14219.108,E2 14219.108} C_VEL
LIN {X 0,Y 458.178,Z 839.06,A -85,B 0,C 180,E1 14230.308,E2 14230.308} C_VEL
LIN {X 0,Y 463.632,Z 846.666,A -85,B 0,C 180,E1 14234.021,E2 14234.021} C_VEL
LIN {X 0,Y 483.77,Z 873.679,A -85,B 0,C 180,E1 14242.537,E2 14242.537} C_VEL
LIN {X 0,Y 509.762,Z 911.546,A -85,B 0,C 180,E1 14249.959,E2 14249.959} C_VEL
LIN {X 0,Y 535.555,Z 961.828,A -85,B 0,C 180,E1 14256.565,E2 14256.565} C_VEL
LIN {X 0,Y 536.257,Z 971.914,A -85,B 0,C 180,E1 14257.211,E2 14257.211} C_VEL
LIN {X 0,Y 521.239,Z 1045.371,A -85,B 0,C 180,E1 14260.536,E2 14260.536} C_VEL
LIN {X 0,Y 502.704,Z 1114.635,A -85,B 0,C 180,E1 14265.706,E2 14265.706} C_VEL
LIN {X 0,Y 484.691,Z 1174.881,A -85,B 0,C 180,E1 14272.652,E2 14272.652} C_VEL
LIN {X 0,Y 470.57,Z 1223.838,A -85,B 0,C 180,E1 14281.159,E2 14281.159} C_VEL
LIN {X 0,Y 462.235,Z 1259.794,A -85,B 0,C 180,E1 14290.827,E2 14290.827} C_VEL
LIN {X 0,Y 459.439,Z 1278.967,A -85,B 0,C 180,E1 14299.53,E2 14299.53} C_VEL
LIN {X 0,Y 459.093,Z 1286.38,A -85,B 0,C 180,E1 14307.157,E2 14307.157} C_VEL
LIN {X 0,Y 459.184,Z 1285.317,A -85,B 0,C 180,E1 14314.777,E2 14314.777} C_VEL
LIN {X 0,Y 451.35,Z 1280.811,A -85,B 0,C 180,E1 14319.111,E2 14319.111} C_VEL
LIN {X 0,Y 454.032,Z 1262.275,A -85,B 0,C 180,E1 14328.521,E2 14328.521} C_VEL
LIN {X 0,Y 461.827,Z 1227.56,A -85,B 0,C 180,E1 14338.467,E2 14338.467} C_VEL
LIN {X 0,Y 476.533,Z 1178.932,A -85,B 0,C 180,E1 14347.335,E2 14347.335} C_VEL
LIN {X 0,Y 495.577,Z 1118.346,A -85,B 0,C 180,E1 14354.581,E2 14354.581} C_VEL
LIN {X 0,Y 514.666,Z 1050.078,A -85,B 0,C 180,E1 14359.857,E2 14359.857} C_VEL
LIN {X 0,Y 530.552,Z 974.809,A -85,B 0,C 180,E1 14363.423,E2 14363.423} C_VEL
LIN {X 0,Y 529.94,Z 964.967,A -85,B 0,C 180,E1 14364.089,E2 14364.089} C_VEL
LIN {X 0,Y 505.163,Z 915.487,A -85,B 0,C 180,E1 14370.793,E2 14370.793} C_VEL
LIN {X 0,Y 481.613,Z 880.772,A -85,B 0,C 180,E1 14377.854,E2 14377.854} C_VEL
LIN {X 0,Y 461.987,Z 854.387,A -85,B 0,C 180,E1 14386.412,E2 14386.412} C_VEL
LIN {X 0,Y 454.582,Z 846.039,A -85,B 0,C 180,E1 14391.79,E2 14391.79} C_VEL
LIN {X 0,Y 451.307,Z 839.06,A -85,B 0,C 180,E1 14398.982,E2 14398.982} C_VEL
LIN {X 0,Y 457.001,Z 848.302,A -85,B 0,C 180,E1 14410.669,E2 14410.669} C_VEL
LIN {X 0,Y 469.309,Z 864.634,A -85,B 0,C 180,E1 14417.784,E2 14417.784} C_VEL
LIN {X 0,Y 490.413,Z 893.447,A -85,B 0,C 180,E1 14425.548,E2 14425.548} C_VEL
LIN {X 0,Y 514.956,Z 936.621,A -85,B 0,C 180,E1 14432.971,E2 14432.971} C_VEL
LIN {X 0,Y 528.256,Z 971.072,A -85,B 0,C 180,E1 14437.294,E2 14437.294} C_VEL
LIN {X 0,Y 511.568,Z 1043.909,A -85,B 0,C 180,E1 14441.251,E2 14441.251} C_VEL
LIN {X 0,Y 492.25,Z 1109.339,A -85,B 0,C 180,E1 14446.972,E2 14446.972} C_VEL
LIN {X 0,Y 473.944,Z 1164.448,A -85,B 0,C 180,E1 14454.349,E2 14454.349} C_VEL
LIN {X 0,Y 460.237,Z 1207.996,A -85,B 0,C 180,E1 14463.271,E2 14463.271} C_VEL
LIN {X 0,Y 453.589,Z 1237.328,A -85,B 0,C 180,E1 14472.814,E2 14472.814} C_VEL
LIN {X 0,Y 451.292,Z 1253.207,A -85,B 0,C 180,E1 14482.217,E2 14482.217} C_VEL
LIN {X 0,Y 451.166,Z 1257.037,A -85,B 0,C 180,E1 14490.963,E2 14490.963} C_VEL
LIN {X 0,Y 451.495,Z 1250.811,A -85,B 0,C 180,E1 14499.678,E2 14499.678} C_VEL
LIN {X 0,Y 453.982,Z 1232.602,A -85,B 0,C 180,E1 14509.028,E2 14509.028} C_VEL
LIN {X 0,Y 461.733,Z 1202.396,A -85,B 0,C 180,E1 14518.054,E2 14518.054} C_VEL
LIN {X 0,Y 476.325,Z 1157.059,A -85,B 0,C 180,E1 14526.758,E2 14526.758} C_VEL
LIN {X 0,Y 495.261,Z 1099.67,A -85,B 0,C 180,E1 14533.955,E2 14533.955} C_VEL
LIN {X 0,Y 514.206,Z 1034.676,A -85,B 0,C 180,E1 14539.246,E2 14539.246} C_VEL
LIN {X 0,Y 527.944,Z 967.363,A -85,B 0,C 180,E1 14542.916,E2 14542.916} C_VEL
LIN {X 0,Y 505.146,Z 917.811,A -85,B 0,C 180,E1 14549.812,E2 14549.812} C_VEL
LIN {X 0,Y 481.44,Z 880.806,A -85,B 0,C 180,E1 14557.287,E2 14557.287} C_VEL
LIN {X 0,Y 462.012,Z 854.245,A -85,B 0,C 180,E1 14565.798,E2 14565.798} C_VEL
LIN {X 0,Y 454.76,Z 846.038,A -85,B 0,C 180,E1 14570.937,E2 14570.937} C_VEL
LIN {X 0,Y 451.297,Z 839.06,A -85,B 0,C 180,E1 14579.092,E2 14579.092} C_VEL
LIN {X 0,Y 451.822,Z 843.392,A -85,B 0,C 180,E1 14585.274,E2 14585.274} C_VEL
LIN {X 0,Y 457.348,Z 849.737,A -85,B 0,C 180,E1 14590.749,E2 14590.749} C_VEL
LIN {X 0,Y 468.707,Z 863.384,A -85,B 0,C 180,E1 14597.144,E2 14597.144} C_VEL
LIN {X 0,Y 492.564,Z 895.841,A -85,B 0,C 180,E1 14605.663,E2 14605.663} C_VEL
LIN {X 0,Y 519.761,Z 942.555,A -85,B 0,C 180,E1 14613.153,E2 14613.153} C_VEL
LIN {X 0,Y 531.299,Z 972.062,A -85,B 0,C 180,E1 14616.526,E2 14616.526} C_VEL
LIN {X 0,Y 515.705,Z 1045.974,A -85,B 0,C 180,E1 14619.896,E2 14619.896} C_VEL
LIN {X 0,Y 496.488,Z 1115.213,A -85,B 0,C 180,E1 14625.115,E2 14625.115} C_VEL
LIN {X 0,Y 478.034,Z 1174.601,A -85,B 0,C 180,E1 14632.04,E2 14632.04} C_VEL
LIN {X 0,Y 463.373,Z 1223.022,A -85,B 0,C 180,E1 14640.537,E2 14640.537} C_VEL
LIN {X 0,Y 454.825,Z 1258.151,A -85,B 0,C 180,E1 14649.994,E2 14649.994} C_VEL
LIN {X 0,Y 451.47,Z 1278.701,A -85,B 0,C 180,E1 14659.343,E2 14659.343} C_VEL
LIN {X 0,Y 451.087,Z 1286.183,A -85,B 0,C 180,E1 14667.107,E2 14667.107} C_VEL
LIN {X 0,Y 451.18,Z 1285.119,A -85,B 0,C 180,E1 14674.826,E2 14674.826} C_VEL
LIN {X 0,Y 451.35,Z 1280.811,A -85,B 0,C 180,E1 14679.111,E2 14679.111} C_VEL
LIN {X 0,Y 443.981,Z 1273.992,A -85,B 0,C 180,E1 14683.49,E2 14683.49} C_VEL
LIN {X 0,Y 447.818,Z 1251.74,A -85,B 0,C 180,E1 14692.42,E2 14692.42} C_VEL
LIN {X 0,Y 457.568,Z 1216.242,A -85,B 0,C 180,E1 14701.389,E2 14701.389} C_VEL
LIN {X 0,Y 474.391,Z 1164.711,A -85,B 0,C 180,E1 14709.944,E2 14709.944} C_VEL
LIN {X 0,Y 494.681,Z 1102.06,A -85,B 0,C 180,E1 14716.729,E2 14716.729} C_VEL
LIN {X 0,Y 513.401,Z 1034.6,A -85,B 0,C 180,E1 14721.422,E2 14721.422} C_VEL
LIN {X 0,Y 525.422,Z 970.865,A -85,B 0,C 180,E1 14724.412,E2 14724.412} C_VEL
LIN {X 0,Y 501.929,Z 922.092,A -85,B 0,C 180,E1 14731.152,E2 14731.152} C_VEL
LIN {X 0,Y 479.297,Z 887.809,A -85,B 0,C 180,E1 14738.231,E2 14738.231} C_VEL
LIN {X 0,Y 460.397,Z 862.088,A -85,B 0,C 180,E1 14746.729,E2 14746.729} C_VEL
